C01810=1075.371,111.105,430.185,173.688,24.346,154.284
C01811=1075.364,110.824,430.206,173.687,24.343,154.284
C01812=1075.358,110.542,430.227,173.684,24.341,154.284
C01813=1075.352,110.293,430.246,173.683,24.338,154.283
C01814=1075.347,110.044,430.266,173.681,24.335,154.283
C01815=1075.341,109.795,430.284,173.680,24.333,154.283
C01816=1075.335,109.546,430.303,173.678,24.330,154.283
C01817=1075.329,109.296,430.322,173.676,24.328,154.282
C01818=1075.323,109.047,430.341,173.675,24.325,154.282
C01819=1075.317,108.798,430.360,173.673,24.323,154.282
C01820=1075.312,108.549,430.379,173.671,24.320,154.282
C01821=1075.306,108.300,430.398,173.670,24.318,154.281
C01822=1075.300,108.050,430.417,173.668,24.316,154.281
C01823=1075.294,107.801,430.436,173.666,24.313,154.281
C01824=1075.289,107.552,430.455,173.665,24.311,154.280
C01825=1075.283,107.302,430.473,173.663,24.308,154.280
C01826=1075.277,107.053,430.492,173.661,24.305,154.280
C01827=1075.272,106.804,430.511,173.660,24.303,154.279
C01828=1075.266,106.555,430.530,173.658,24.300,154.279
C01829=1075.260,106.306,430.549,173.656,24.298,154.279
C01830=1075.255,106.056,430.568,173.655,24.295,154.279
C01831=1075.249,105.808,430.587,173.653,24.293,154.278
C01832=1075.243,105.558,430.605,173.651,24.290,154.278
C01833=1075.237,105.309,430.624,173.650,24.287,154.278
C01834=1075.232,105.060,430.643,173.649,24.285,154.277
C01835=1075.226,104.811,430.662,173.646,24.282,154.277
C01836=1075.220,104.561,430.680,173.645,24.280,154.277
C01837=1075.215,104.312,430.699,173.644,24.277,154.277
C01838=1075.209,104.063,430.718,173.642,24.275,154.276
C01839=1075.203,103.814,430.737,173.640,24.272,154.276
C01840=1075.198,103.565,430.756,173.639,24.269,154.276
C01841=1075.192,103.315,430.774,173.637,24.267,154.275
C01842=1075.186,103.066,430.793,173.635,24.264,154.275
C01843=1075.181,102.817,430.812,173.634,24.262,154.275
C01844=1075.175,102.567,430.830,173.632,24.260,154.274
C01845=1075.169,102.318,430.849,173.630,24.256,154.274
C01846=1075.164,102.069,430.868,173.629,24.254,154.274
C01847=1075.158,101.820,430.886,173.627,24.252,154.274
C01848=1075.153,101.571,430.904,173.625,24.249,154.273
C01849=1075.146,101.321,430.923,173.624,24.247,154.273
C01850=1075.141,101.071,430.942,173.623,24.244,154.273
C01851=1075.135,100.823,430.960,173.621,24.241,154.272
C01852=1075.129,100.574,430.979,173.619,24.239,154.272
C01853=1075.123,100.324,430.997,173.618,24.236,154.272
C01854=1075.118,100.075,431.016,173.616,24.234,154.271
C01855=1075.112,99.826,431.035,173.614,24.231,154.271
C01856=1075.106,99.576,431.053,173.613,24.229,154.271
C01857=1075.101,99.327,431.071,173.611,24.227,154.271
C01858=1075.095,99.078,431.089,173.609,24.224,154.270
C01859=1075.089,98.828,431.109,173.608,24.221,154.270
C01860=1075.083,98.580,431.127,173.606,24.219,154.270
C01861=1075.077,98.330,431.145,173.605,24.216,154.269
C01862=1075.072,98.081,431.164,173.603,24.213,154.269
C01863=1075.066,97.832,431.182,173.602,24.211,154.269
C01864=1075.060,97.582,431.201,173.600,24.209,154.269
C01865=1075.054,97.333,431.218,173.598,24.206,154.268
C01866=1075.048,97.084,431.237,173.597,24.203,154.268
C01867=1075.043,96.835,431.255,173.595,24.201,154.268
C01868=1075.037,96.586,431.274,173.593,24.198,154.267
C01869=1075.031,96.336,431.292,173.592,24.196,154.267
C01870=1075.026,96.087,431.311,173.590,24.193,154.267
C01871=1075.019,95.837,431.329,173.589,24.191,154.266
C01872=1075.014,95.589,431.348,173.587,24.188,154.266
C01873=1075.008,95.307,431.368,173.586,24.185,154.266
C01874=1075.001,95.025,431.388,173.583,24.182,154.265
C01875=1074.995,94.744,431.409,173.582,24.180,154.265
C01876=1074.988,94.462,431.430,173.580,24.176,154.265
C01877=1074.983,94.213,431.449,173.579,24.174,154.264
C01878=1074.977,93.963,431.467,173.576,24.171,154.264
C01879=1074.971,93.714,431.484,173.575,24.168,154.264
C01880=1074.965,93.465,431.503,173.574,24.166,154.263
C01881=1074.960,93.216,431.521,173.572,24.164,154.263
C01882=1074.953,92.967,431.540,173.570,24.161,154.263
C01883=1074.949,92.717,431.558,173.569,24.159,154.263
C01884=1074.943,92.468,431.576,173.568,24.156,154.262
C01885=1074.937,92.219,431.594,173.566,24.153,154.262
C01886=1074.931,91.970,431.612,173.564,24.151,154.262
C01887=1074.926,91.720,431.630,173.563,24.148,154.261
C01888=1074.919,91.471,431.649,173.561,24.145,154.261
C01889=1074.914,91.222,431.666,173.559,24.143,154.261
C01890=1074.909,90.972,431.685,173.558,24.140,154.260
C01891=1074.903,90.724,431.703,173.556,24.138,154.260
C01892=1074.897,90.474,431.721,173.555,24.136,154.260
C01893=1074.891,90.225,431.739,173.553,24.132,154.259
C01894=1074.885,89.975,431.757,173.552,24.130,154.259
C01895=1074.879,89.727,431.775,173.550,24.128,154.259
C01896=1074.874,89.477,431.793,173.549,24.125,154.259
C01897=1074.868,89.228,431.811,173.547,24.122,154.258
C01898=1074.862,88.978,431.829,173.545,24.120,154.258
C01899=1074.856,88.729,431.847,173.544,24.117,154.258
C01900=1074.850,88.480,431.865,173.543,24.115,154.257
C01901=1074.844,88.230,431.883,173.541,24.112,154.257
C01902=1074.839,87.981,431.901,173.539,24.110,154.257
C01903=1074.833,87.732,431.919,173.538,24.107,154.257
C01904=1074.827,87.483,431.937,173.537,24.105,154.256
C01905=1074.821,87.234,431.954,173.534,24.102,154.256
C01906=1074.815,86.984,431.972,173.533,24.099,154.256
C01907=1074.810,86.735,431.990,173.532,24.097,154.255
C01908=1074.804,86.485,432.008,173.530,24.095,154.255
C01909=1074.798,86.236,432.027,173.528,24.092,154.255
C01910=1074.792,85.987,432.045,173.527,24.089,154.254
C01911=1074.787,85.738,432.062,173.526,24.087,154.254
C01912=1074.780,85.488,432.080,173.524,24.084,154.254
C01913=1074.775,85.239,432.098,173.522,24.081,154.254
C01914=1074.769,84.989,432.116,173.521,24.079,154.253
C01915=1074.763,84.740,432.133,173.519,24.076,154.253
C01916=1074.758,84.491,432.151,173.518,24.074,154.253
C01917=1074.752,84.241,432.169,173.516,24.071,154.252
C01918=1074.746,83.992,432.186,173.514,24.069,154.252
C01919=1074.740,83.743,432.205,173.513,24.066,154.252
C01920=1074.734,83.494,432.222,173.512,24.063,154.251
C01921=1074.729,83.245,432.240,173.510,24.061,154.251
C01922=1074.723,82.995,432.258,173.508,24.058,154.251
C01923=1074.717,82.746,432.275,173.507,24.056,154.250
C01924=1074.711,82.497,432.293,173.506,24.053,154.250
C01925=1074.705,82.247,432.311,173.504,24.050,154.250
C01926=1074.700,81.998,432.329,173.502,24.048,154.249
C01927=1074.694,81.749,432.346,173.501,24.046,154.249
C01928=1074.688,81.500,432.364,173.500,24.043,154.249
C01929=1074.683,81.251,432.382,173.497,24.040,154.249
C01930=1074.677,81.001,432.400,173.496,24.038,154.248
C01931=1074.671,80.752,432.417,173.495,24.035,154.248
C01932=1074.666,80.503,432.435,173.494,24.032,154.248
C01933=1074.659,80.253,432.453,173.491,24.030,154.247
C01934=1074.654,80.003,432.469,173.490,24.027,154.247
C01935=1074.649,79.754,432.487,173.489,24.024,154.247
C01936=1074.643,79.505,432.505,173.487,24.022,154.246
C01937=1074.636,79.224,432.525,173.485,24.019,154.246
C01938=1074.630,78.942,432.545,173.484,24.016,154.246
C01939=1074.624,78.661,432.565,173.482,24.013,154.245
C01940=1074.617,78.379,432.585,173.481,24.010,154.245
C01941=1074.612,78.129,432.602,173.478,24.007,154.245
C01942=1074.606,77.880,432.620,173.477,24.005,154.244
C01943=1074.600,77.631,432.637,173.476,24.003,154.244
C01944=1074.594,77.382,432.654,173.475,24.000,154.244
C01945=1074.588,77.132,432.672,173.472,23.997,154.243
C01946=1074.582,76.883,432.690,173.471,23.994,154.243
C01947=1074.577,76.634,432.708,173.470,23.992,154.243
C01948=1074.571,76.384,432.725,173.469,23.989,154.242
C01949=1074.564,76.135,432.742,173.467,23.987,154.242
C01950=1074.559,75.886,432.759,173.465,23.984,154.242
C01951=1074.553,75.637,432.777,173.464,23.982,154.242
C01952=1074.547,75.387,432.795,173.462,23.979,154.241
C01953=1074.542,75.137,432.812,173.461,23.976,154.241
C01954=1074.536,74.889,432.829,173.459,23.974,154.241
C01955=1074.530,74.639,432.847,173.457,23.971,154.240
C01956=1074.524,74.390,432.864,173.456,23.969,154.240
C01957=1074.519,74.140,432.881,173.455,23.966,154.240
C01958=1074.512,73.891,432.898,173.454,23.964,154.239
C01959=1074.507,73.642,432.916,173.451,23.961,154.239
C01960=1074.501,73.392,432.933,173.450,23.958,154.239
C01961=1074.496,73.143,432.950,173.449,23.956,154.238
C01962=1074.489,72.894,432.968,173.448,23.953,154.238
C01963=1074.483,72.645,432.985,173.446,23.951,154.238
C01964=1074.478,72.395,433.002,173.444,23.948,154.237
C01965=1074.473,72.146,433.020,173.443,23.945,154.237
C01966=1074.466,71.897,433.037,173.441,23.943,154.237
C01967=1074.461,71.647,433.054,173.440,23.940,154.237
C01968=1074.455,71.398,433.071,173.438,23.937,154.236
C01969=1074.449,71.149,433.088,173.437,23.935,154.236
C01970=1074.443,70.899,433.106,173.435,23.932,154.236
C01971=1074.438,70.650,433.123,173.434,23.930,154.235
C01972=1074.432,70.400,433.140,173.433,23.927,154.235
C01973=1074.426,70.151,433.157,173.431,23.924,154.235
C01974=1074.420,69.902,433.175,173.429,23.922,154.234
C01975=1074.414,69.652,433.191,173.428,23.919,154.234
C01976=1074.408,69.403,433.209,173.427,23.917,154.234
C01977=1074.403,69.154,433.226,173.425,23.914,154.233
C01978=1074.396,68.904,433.243,173.423,23.911,154.233
C01979=1074.391,68.655,433.260,173.422,23.909,154.233
C01980=1074.386,68.405,433.277,173.421,23.906,154.232
C01981=1074.379,68.157,433.294,173.419,23.904,154.232
C01982=1074.374,67.907,433.311,173.418,23.901,154.232
C01983=1074.367,67.658,433.328,173.416,23.898,154.231
C01984=1074.362,67.408,433.345,173.415,23.896,154.231
C01985=1074.356,67.159,433.362,173.413,23.893,154.231
C01986=1074.351,66.910,433.379,173.412,23.891,154.231
C01987=1074.345,66.660,433.397,173.411,23.888,154.230
C01988=1074.339,66.410,433.413,173.408,23.885,154.230
C01989=1074.333,66.161,433.431,173.407,23.883,154.230
C01990=1074.327,65.912,433.447,173.406,23.881,154.229
C01991=1074.322,65.663,433.465,173.405,23.878,154.229
C01992=1074.316,65.414,433.481,173.403,23.875,154.229
C01993=1074.310,65.163,433.498,173.401,23.872,154.228
C01994=1074.304,64.915,433.515,173.400,23.870,154.228
C01995=1074.298,64.665,433.532,173.399,23.867,154.228
C01996=1074.292,64.416,433.549,173.397,23.865,154.227
C01997=1074.287,64.167,433.566,173.396,23.862,154.227
C01998=1074.281,63.918,433.583,173.394,23.860,154.227
C01999=1074.274,63.668,433.599,173.392,23.857,154.226
C02000=1074.269,63.418,433.616,173.391,23.854,154.226
C02001=1074.262,63.137,433.635,173.389,23.852,154.226
C02002=1074.255,62.855,433.654,173.388,23.849,154.226
C02003=1074.248,62.574,433.673,173.386,23.846,154.225
C02004=1074.242,62.293,433.692,173.384,23.843,154.225
C02005=1074.236,62.042,433.709,173.383,23.841,154.225
C02006=1074.230,61.793,433.726,173.382,23.838,154.224
C02007=1074.224,61.544,433.742,173.380,23.835,154.224
C02008=1074.218,61.294,433.759,173.378,23.833,154.224
C02009=1074.212,61.046,433.776,173.377,23.830,154.223
C02010=1074.206,60.796,433.792,173.376,23.828,154.223
C02011=1074.200,60.546,433.809,173.374,23.825,154.223
C02012=1074.194,60.297,433.826,173.373,23.822,154.222
C02013=1074.188,60.048,433.843,173.371,23.820,154.222
C02014=1074.182,59.799,433.859,173.370,23.817,154.222
C02015=1074.177,59.549,433.876,173.368,23.815,154.222
C02016=1074.171,59.300,433.893,173.367,23.812,154.221
C02017=1074.164,59.050,433.909,173.366,23.810,154.221
C02018=1074.159,58.800,433.926,173.364,23.807,154.221
C02019=1074.153,58.551,433.942,173.362,23.804,154.220
C02020=1074.147,58.302,433.959,173.361,23.802,154.220
C02021=1074.141,58.053,433.976,173.360,23.799,154.220
C02022=1074.136,57.803,433.992,173.358,23.797,154.219
C02023=1074.130,57.554,434.009,173.357,23.794,154.219
C02024=1074.124,57.305,434.025,173.355,23.792,154.219
C02025=1074.118,57.055,434.041,173.354,23.789,154.218
C02026=1074.112,56.806,434.059,173.352,23.786,154.218
C02027=1074.106,56.556,434.075,173.351,23.784,154.218
C02028=1074.100,56.307,434.092,173.350,23.781,154.217
C02029=1074.094,56.058,434.108,173.348,23.778,154.217
C02030=1074.089,55.808,434.125,173.346,23.776,154.217
C02031=1074.083,55.559,434.141,173.345,23.773,154.217
C02032=1074.077,55.309,434.157,173.344,23.771,154.216
C02033=1074.070,55.060,434.174,173.342,23.768,154.216
C02034=1074.065,54.811,434.191,173.341,23.766,154.216
C02035=1074.059,54.561,434.207,173.339,23.763,154.215
C02036=1074.053,54.312,434.224,173.338,23.761,154.215
C02037=1074.047,54.063,434.240,173.336,23.758,154.215
C02038=1074.041,53.813,434.256,173.335,23.755,154.214
C02039=1074.036,53.564,434.273,173.334,23.753,154.214
C02040=1074.030,53.314,434.289,173.333,23.750,154.214
C02041=1074.024,53.065,434.305,173.330,23.747,154.213
C02042=1074.018,52.816,434.322,173.329,23.745,154.213
C02043=1074.012,52.566,434.338,173.328,23.742,154.213
C02044=1074.007,52.317,434.355,173.327,23.739,154.212
C02045=1074.001,52.067,434.371,173.325,23.737,154.212
C02046=1073.995,51.818,434.387,173.323,23.734,154.212
C02047=1073.989,51.569,434.404,173.322,23.731,154.211
C02048=1073.983,51.319,434.420,173.321,23.729,154.211
C02049=1073.978,51.070,434.437,173.319,23.727,154.211
C02050=1073.972,50.820,434.453,173.318,23.724,154.210
C02051=1073.966,50.571,434.469,173.317,23.721,154.210
C02052=1073.960,50.322,434.485,173.315,23.718,154.210
C02053=1073.954,50.072,434.502,173.313,23.716,154.210
C02054=1073.949,49.823,434.519,173.312,23.713,154.209
C02055=1073.943,49.573,434.535,173.311,23.711,154.209
C02056=1073.937,49.324,434.551,173.309,23.708,154.209
C02057=1073.931,49.075,434.567,173.308,23.705,154.208
C02058=1073.925,48.825,434.584,173.306,23.703,154.208
C02059=1073.919,48.576,434.600,173.305,23.700,154.208
C02060=1073.914,48.327,434.616,173.304,23.697,154.207
C02061=1073.909,48.078,434.633,173.302,23.695,154.207
C02062=1073.903,47.828,434.648,173.301,23.693,154.207
C02063=1073.897,47.578,434.664,173.300,23.690,154.206
C02064=1073.891,47.329,434.681,173.298,23.687,154.206
C02065=1073.885,47.047,434.699,173.296,23.684,154.206
C02066=1073.878,46.766,434.717,173.295,23.681,154.205
C02067=1073.871,46.483,434.736,173.293,23.678,154.205
C02068=1073.865,46.202,434.754,173.292,23.675,154.205
C02069=1073.859,45.952,434.770,173.291,23.673,154.204
C02070=1073.854,45.703,434.787,173.288,23.669,154.204
C02071=1073.848,45.454,434.803,173.287,23.667,154.204
C02072=1073.843,45.204,434.818,173.286,23.664,154.203
C02073=1073.837,44.955,434.835,173.285,23.662,154.203
C02074=1073.831,44.705,434.851,173.283,23.659,154.203
C02075=1073.825,44.456,434.867,173.282,23.656,154.202
C02076=1073.819,44.206,434.883,173.280,23.654,154.202
C02077=1073.813,43.957,434.899,173.279,23.651,154.202
C02078=1073.808,43.708,434.915,173.278,23.648,154.201
C02079=1073.802,43.459,434.931,173.276,23.646,154.201
C02080=1073.796,43.209,434.947,173.275,23.644,154.201
C02081=1073.790,42.959,434.963,173.274,23.641,154.200
C02082=1073.785,42.710,434.979,173.272,23.638,154.200
C02083=1073.779,42.461,434.995,173.270,23.635,154.200
C02084=1073.773,42.211,435.011,173.269,23.633,154.199
C02085=1073.767,41.961,435.027,173.268,23.631,154.199
C02086=1073.761,41.712,435.043,173.266,23.628,154.199
C02087=1073.756,41.463,435.059,173.265,23.625,154.198
C02088=1073.750,41.213,435.075,173.264,23.623,154.198
C02089=1073.743,40.964,435.090,173.262,23.620,154.198
C02090=1073.738,40.714,435.106,173.260,23.617,154.198
C02091=1073.732,40.465,435.122,173.259,23.615,154.197
C02092=1073.726,40.216,435.139,173.258,23.612,154.197
C02093=1073.721,39.966,435.154,173.257,23.609,154.197
C02094=1073.715,39.717,435.170,173.255,23.607,154.196
C02095=1073.709,39.467,435.186,173.254,23.605,154.196
C02096=1073.703,39.218,435.202,173.252,23.601,154.196
C02097=1073.697,38.968,435.218,173.251,23.599,154.195
C02098=1073.691,38.719,435.233,173.249,23.596,154.195
C02099=1073.686,38.470,435.249,173.248,23.594,154.195
C02100=1073.680,38.220,435.264,173.247,23.591,154.194
C02101=1073.674,37.971,435.281,173.246,23.589,154.194
C02102=1073.668,37.721,435.297,173.244,23.586,154.194
C02103=1073.662,37.471,435.312,173.242,23.584,154.194
C02104=1073.656,37.222,435.328,173.241,23.581,154.193
C02105=1073.651,36.973,435.343,173.240,23.578,154.193
C02106=1073.645,36.724,435.360,173.238,23.576,154.193
C02107=1073.638,36.474,435.375,173.237,23.573,154.192
C02108=1073.632,36.225,435.391,173.236,23.570,154.192
C02109=1073.627,35.975,435.406,173.234,23.568,154.192
C02110=1073.621,35.726,435.422,173.232,23.565,154.191
C02111=1073.615,35.476,435.437,173.231,23.563,154.191
C02112=1073.609,35.227,435.453,173.230,23.560,154.191
C02113=1073.603,34.977,435.469,173.229,23.558,154.190
C02114=1073.597,34.728,435.485,173.227,23.555,154.190
C02115=1073.592,34.479,435.500,173.226,23.553,154.190
C02116=1073.586,34.229,435.516,173.224,23.550,154.189
C02117=1073.579,33.980,435.531,173.222,23.548,154.189
C02118=1073.574,33.730,435.547,173.221,23.545,154.189
C02119=1073.568,33.480,435.563,173.220,23.542,154.189
C02120=1073.562,33.232,435.577,173.219,23.540,154.188
C02121=1073.556,32.982,435.594,173.217,23.537,154.188
C02122=1073.550,32.732,435.609,173.216,23.534,154.188
C02123=1073.544,32.483,435.624,173.214,23.532,154.187
C02124=1073.539,32.234,435.640,173.213,23.529,154.187
C02125=1073.533,31.984,435.656,173.211,23.527,154.187
C02126=1073.526,31.735,435.671,173.210,23.524,154.186
C02127=1073.521,31.485,435.687,173.209,23.521,154.186
C02128=1073.516,31.236,435.702,173.208,23.519,154.186
C02129=1073.508,30.954,435.719,173.206,23.516,154.185
C02130=1073.502,30.672,435.737,173.204,23.513,154.185
C02131=1073.495,30.390,435.754,173.203,23.510,154.185
C02132=1073.489,30.108,435.772,173.201,23.507,154.184
C02133=1073.483,29.859,435.787,173.200,23.505,154.184
C02134=1073.477,29.609,435.803,173.199,23.502,154.184
C02135=1073.471,29.360,435.818,173.197,23.499,154.183
C02136=1073.465,29.110,435.833,173.196,23.497,154.183
C02137=1073.459,28.861,435.850,173.194,23.494,154.183
C02138=1073.453,28.612,435.864,173.193,23.492,154.182
C02139=1073.448,28.362,435.880,173.191,23.489,154.182
C02140=1073.441,28.112,435.895,173.190,23.486,154.182
C02141=1073.436,27.864,435.911,173.189,23.484,154.182
C02142=1073.430,27.614,435.926,173.188,23.482,154.181
C02143=1073.424,27.364,435.941,173.186,23.479,154.181
C02144=1073.418,27.115,435.956,173.185,23.477,154.181
C02145=1073.413,26.865,435.971,173.183,23.473,154.180
C02146=1073.406,26.616,435.987,173.182,23.471,154.180
C02147=1073.400,26.366,436.002,173.180,23.469,154.180
C02148=1073.394,26.117,436.017,173.179,23.466,154.179
C02149=1073.389,25.867,436.033,173.178,23.464,154.179
C02150=1073.382,25.618,436.047,173.176,23.461,154.179
C02151=1073.376,25.369,436.063,173.175,23.458,154.178
C02152=1073.371,25.119,436.078,173.173,23.456,154.178
C02153=1073.364,24.870,436.093,173.172,23.453,154.178
C02154=1073.359,24.620,436.108,173.170,23.451,154.178
C02155=1073.353,24.371,436.123,173.169,23.448,154.177
C02156=1073.347,24.121,436.139,173.168,23.445,154.177
C02157=1073.342,23.872,436.153,173.167,23.443,154.177
C02158=1073.335,23.623,436.169,173.165,23.441,154.176
C02159=1073.329,23.373,436.185,173.164,23.438,154.176
C02160=1073.323,23.124,436.199,173.162,23.435,154.176
C02161=1073.318,22.874,436.215,173.161,23.433,154.176
C02162=1073.311,22.624,436.230,173.159,23.430,154.175
C02163=1073.306,22.375,436.245,173.158,23.428,154.175
C02164=1073.300,22.125,436.260,173.157,23.425,154.175
C02165=1073.294,21.876,436.274,173.156,23.423,154.174
C02166=1073.289,21.626,436.290,173.154,23.420,154.174
C02167=1073.282,21.377,436.305,173.153,23.417,154.174
C02168=1073.277,21.128,436.320,173.151,23.415,154.173
C02169=1073.271,20.878,436.335,173.150,23.412,154.173
C02170=1073.264,20.628,436.350,173.148,23.410,154.173
C02171=1073.259,20.379,436.365,173.147,23.407,154.172
C02172=1073.253,20.129,436.380,173.146,23.404,154.172
C02173=1073.247,19.880,436.395,173.145,23.402,154.172
C02174=1073.241,19.630,436.410,173.143,23.400,154.172
C02175=1073.235,19.381,436.425,173.142,23.397,154.171
C02176=1073.229,19.132,436.440,173.140,23.394,154.171
C02177=1073.223,18.882,436.455,173.138,23.392,154.171
C02178=1073.218,18.633,436.470,173.137,23.390,154.170
C02179=1073.211,18.383,436.485,173.136,23.387,154.170
C02180=1073.205,18.134,436.500,173.135,23.384,154.170
C02181=1073.200,17.884,436.515,173.133,23.382,154.169
C02182=1073.194,17.635,436.530,173.132,23.379,154.169
C02183=1073.188,17.386,436.544,173.131,23.377,154.169
C02184=1073.182,17.136,436.559,173.129,23.374,154.169
C02185=1073.176,16.887,436.575,173.127,23.372,154.168
C02186=1073.170,16.637,436.590,173.126,23.369,154.168
C02187=1073.165,16.387,436.603,173.125,23.366,154.168
C02188=1073.158,16.138,436.618,173.124,23.364,154.167
C02189=1073.153,15.888,436.634,173.122,23.362,154.167
C02190=1073.147,15.639,436.648,173.121,23.359,154.167
C02191=1073.140,15.389,436.663,173.120,23.357,154.167
C02192=1073.135,15.140,436.678,173.118,23.353,154.166
C02193=1073.128,14.860,436.695,173.116,23.351,154.166
C02194=1073.121,14.580,436.711,173.115,23.348,154.165
C02195=1073.115,14.299,436.728,173.113,23.345,154.165
C02196=1073.108,14.018,436.745,173.112,23.342,154.165
C02197=1073.102,13.769,436.759,173.111,23.340,154.165
C02198=1073.096,13.519,436.773,173.109,23.337,154.164
C02199=1073.090,13.270,436.788,173.108,23.335,154.164
C02200=1073.084,13.021,436.803,173.106,23.332,154.164
C02201=1073.078,12.770,436.818,173.105,23.330,154.163
C02202=1073.073,12.521,436.832,173.103,23.327,154.163
C02203=1073.066,12.271,436.847,173.102,23.325,154.163
C02204=1073.060,12.022,436.862,173.101,23.323,154.163
C02205=1073.054,11.772,436.876,173.099,23.320,154.162
C02206=1073.049,11.523,436.891,173.098,23.318,154.162
C02207=1073.042,11.274,436.906,173.097,23.315,154.162
C02208=1073.036,11.025,436.920,173.096,23.313,154.161
C02209=1073.030,10.774,436.934,173.093,23.310,154.161
C02210=1073.025,10.525,436.949,173.092,23.308,154.161
C02211=1073.018,10.276,436.964,173.091,23.305,154.161
C02212=1073.013,10.026,436.978,173.090,23.303,154.160
C02213=1073.006,9.776,436.993,173.088,23.300,154.160
C02214=1073.001,9.528,437.007,173.087,23.298,154.160
C02215=1072.994,9.277,437.022,173.086,23.296,154.159
C02216=1072.989,9.028,437.036,173.084,23.293,154.159
C02217=1072.982,8.779,437.051,173.082,23.290,154.159
C02218=1072.977,8.529,437.065,173.081,23.287,154.159
C02219=1072.970,8.279,437.080,173.080,23.285,154.158
C02220=1072.965,8.030,437.095,173.078,23.283,154.158
C02221=1072.959,7.780,437.109,173.077,23.280,154.158
C02222=1072.953,7.531,437.123,173.076,23.278,154.157
C02223=1072.946,7.282,437.138,173.075,23.275,154.157
C02224=1072.941,7.032,437.152,173.073,23.273,154.157
C02225=1072.935,6.782,437.167,173.072,23.270,154.157
C02226=1072.929,6.533,437.181,173.070,23.268,154.156
C02227=1072.923,6.283,437.196,173.069,23.265,154.156
C02228=1072.917,6.034,437.210,173.067,23.263,154.156
C02229=1072.911,5.785,437.224,173.066,23.260,154.155
C02230=1072.905,5.535,437.239,173.065,23.258,154.155
C02231=1072.900,5.285,437.253,173.063,23.255,154.155
C02232=1072.893,5.036,437.268,173.062,23.253,154.155
C02233=1072.888,4.786,437.282,173.061,23.251,154.154
C02234=1072.881,4.537,437.296,173.059,23.248,154.154
C02235=1072.875,4.287,437.310,173.057,23.245,154.154
C02236=1072.869,4.038,437.325,173.056,23.242,154.153
C02237=1072.863,3.788,437.339,173.055,23.240,154.153
C02238=1072.857,3.539,437.354,173.054,23.238,154.153
C02239=1072.852,3.289,437.367,173.052,23.235,154.153
C02240=1072.846,3.040,437.382,173.051,23.233,154.152
C02241=1072.840,2.790,437.396,173.050,23.230,154.152
C02242=1072.834,2.541,437.411,173.049,23.228,154.152
C02243=1072.828,2.291,437.425,173.046,23.225,154.151
C02244=1072.823,2.041,437.439,173.045,23.223,154.151
C02245=1072.816,1.792,437.454,173.044,23.220,154.151
C02246=1072.811,1.542,437.468,173.042,23.218,154.151
C02247=1072.805,1.293,437.482,173.041,23.215,154.150
C02248=1072.798,1.043,437.496,173.040,23.213,154.150
C02249=1072.793,0.794,437.511,173.039,23.211,154.150
C02250=1072.787,0.545,437.524,173.037,23.208,154.149
C02251=1072.781,0.294,437.539,173.036,23.206,154.149
C02252=1072.775,0.045,437.553,173.034,23.203,154.149
C02253=1072.770,-0.204,437.567,173.033,23.200,154.149
C02254=1072.764,-0.454,437.581,173.031,23.198,154.148
C02255=1072.758,-0.703,437.596,173.030,23.196,154.148
C02256=1072.752,-0.953,437.610,173.029,23.193,154.148
C02257=1072.745,-1.231,437.626,173.028,23.190,154.147
C02258=1072.739,-1.510,437.641,173.025,23.187,154.147
C02259=1072.732,-1.788,437.657,173.024,23.184,154.147
C02260=1072.726,-2.067,437.673,173.023,23.182,154.146
C02261=1072.720,-2.316,437.687,173.021,23.179,154.146
C02262=1072.714,-2.565,437.701,173.020,23.177,154.146
C02263=1072.709,-2.815,437.715,173.018,23.174,154.146
C02264=1072.702,-3.065,437.730,173.017,23.172,154.145
C02265=1072.697,-3.314,437.743,173.016,23.170,154.145
C02266=1072.691,-3.564,437.757,173.014,23.167,154.145
C02267=1072.685,-3.814,437.771,173.013,23.165,154.145
C02268=1072.679,-4.063,437.785,173.012,23.162,154.144
C02269=1072.673,-4.312,437.799,173.011,23.160,154.144
C02270=1072.667,-4.562,437.813,173.009,23.157,154.144
C02271=1072.661,-4.812,437.827,173.007,23.155,154.143
C02272=1072.655,-5.061,437.841,173.006,23.152,154.143
C02273=1072.648,-5.311,437.855,173.004,23.150,154.143
C02274=1072.643,-5.560,437.869,173.003,23.148,154.143
C02275=1072.637,-5.810,437.882,173.002,23.145,154.142
C02276=1072.631,-6.060,437.896,173.001,23.143,154.142
C02277=1072.625,-6.309,437.911,172.999,23.141,154.142
C02278=1072.619,-6.558,437.924,172.998,23.138,154.142
C02279=1072.613,-6.808,437.938,172.997,23.136,154.141
C02280=1072.606,-7.058,437.952,172.995,23.133,154.141
C02281=1072.601,-7.307,437.966,172.993,23.130,154.141
C02282=1072.595,-7.557,437.980,172.992,23.129,154.141
C02283=1072.588,-7.806,437.994,172.991,23.126,154.140
C02284=1072.583,-8.056,438.008,172.989,23.124,154.140
C02285=1072.577,-8.305,438.021,172.988,23.121,154.140
C02286=1072.571,-8.555,438.035,172.987,23.119,154.140
C02287=1072.565,-8.805,438.049,172.985,23.116,154.139
C02288=1072.559,-9.054,438.062,172.984,23.114,154.139
C02289=1072.553,-9.304,438.076,172.982,23.111,154.139
C02290=1072.547,-9.553,438.089,172.981,23.109,154.138
C02291=1072.541,-9.803,438.104,172.979,23.107,154.138
C02292=1072.535,-10.053,438.117,172.978,23.104,154.138
C02293=1072.529,-10.302,438.131,172.977,23.102,154.138
C02294=1072.524,-10.551,438.145,172.975,23.100,154.137
C02295=1072.517,-10.800,438.159,172.974,23.097,154.137
C02296=1072.511,-11.051,438.173,172.973,23.095,154.137
C02297=1072.505,-11.300,438.186,172.972,23.092,154.137
C02298=1072.500,-11.549,438.200,172.969,23.089,154.136
C02299=1072.493,-11.799,438.213,172.968,23.088,154.136
C02300=1072.488,-12.048,438.227,172.967,23.085,154.136
C02301=1072.481,-12.298,438.241,172.965,23.083,154.136
C02302=1072.476,-12.548,438.255,172.964,23.080,154.135
C02303=1072.470,-12.797,438.269,172.963,23.078,154.135
C02304=1072.464,-13.047,438.282,172.962,23.075,154.135
C02305=1072.458,-13.296,438.296,172.960,23.073,154.135
C02306=1072.452,-13.545,438.309,172.959,23.071,154.134
C02307=1072.446,-13.796,438.323,172.958,23.069,154.134
C02308=1072.440,-14.045,438.336,172.955,23.066,154.134
C02309=1072.435,-14.295,438.350,172.954,23.063,154.134
C02310=1072.429,-14.544,438.363,172.953,23.061,154.133
C02311=1072.423,-14.794,438.377,172.952,23.059,154.133
C02312=1072.417,-15.043,438.390,172.950,23.056,154.133
C02313=1072.411,-15.293,438.404,172.949,23.054,154.133
C02314=1072.405,-15.543,438.418,172.948,23.052,154.132
C02315=1072.398,-15.792,438.431,172.946,23.049,154.132
C02316=1072.393,-16.042,438.445,172.945,23.047,154.132
C02317=1072.387,-16.291,438.458,172.944,23.045,154.132
C02318=1072.380,-16.540,438.471,172.941,23.042,154.131
C02319=1072.374,-16.791,438.485,172.940,23.040,154.131
C02320=1072.369,-17.040,438.498,172.939,23.037,154.131
C02321=1072.362,-17.317,438.512,172.938,23.035,154.130
C02322=1072.355,-17.594,438.528,172.936,23.032,154.130
C02323=1072.349,-17.871,438.542,172.934,23.030,154.130
C02324=1072.342,-18.148,438.557,172.933,23.027,154.130
C02325=1072.336,-18.397,438.571,172.932,23.025,154.130
C02326=1072.330,-18.646,438.584,172.930,23.023,154.129
C02327=1072.324,-18.896,438.598,172.929,23.020,154.129
C02328=1072.318,-19.145,438.612,172.927,23.018,154.129
C02329=1072.312,-19.395,438.624,172.925,23.016,154.129
C02330=1072.306,-19.644,438.637,172.924,23.013,154.128
C02331=1072.301,-19.894,438.651,172.923,23.011,154.128
C02332=1072.294,-20.144,438.665,172.922,23.008,154.128
C02333=1072.288,-20.394,438.678,172.920,23.007,154.128
C02334=1072.282,-20.643,438.691,172.919,23.004,154.127
C02335=1072.276,-20.893,438.705,172.918,23.002,154.127
C02336=1072.270,-21.142,438.718,172.916,23.000,154.127
C02337=1072.264,-21.392,438.730,172.915,22.997,154.127
C02338=1072.259,-21.641,438.744,172.913,22.995,154.126
C02339=1072.252,-21.891,438.758,172.911,22.992,154.126
C02340=1072.246,-22.141,438.770,172.910,22.990,154.126
C02341=1072.240,-22.390,438.783,172.909,22.988,154.126
C02342=1072.235,-22.639,438.797,172.907,22.985,154.125
C02343=1072.229,-22.889,438.811,172.906,22.983,154.125
C02344=1072.222,-23.139,438.823,172.905,22.981,154.125
C02345=1072.216,-23.389,438.837,172.903,22.979,154.125
C02346=1072.210,-23.638,438.851,172.902,22.976,154.124
C02347=1072.204,-23.888,438.863,172.901,22.974,154.124
C02348=1072.198,-24.137,438.876,172.899,22.971,154.124
C02349=1072.192,-24.387,438.889,172.897,22.969,154.124
C02350=1072.187,-24.637,438.903,172.896,22.967,154.124
C02351=1072.181,-24.886,438.916,172.895,22.965,154.123
C02352=1072.175,-25.136,438.929,172.893,22.962,154.123
C02353=1072.168,-25.385,438.942,172.892,22.960,154.123
C02354=1072.163,-25.635,438.956,172.891,22.958,154.123
C02355=1072.157,-25.885,438.968,172.889,22.955,154.122
C02356=1072.151,-26.134,438.982,172.888,22.954,154.122
C02357=1072.145,-26.384,438.994,172.887,22.951,154.122
C02358=1072.140,-26.633,439.008,172.884,22.948,154.122
C02359=1072.134,-26.883,439.021,172.883,22.946,154.121
C02360=1072.127,-27.132,439.034,172.882,22.944,154.121
C02361=1072.121,-27.382,439.047,172.881,22.942,154.121
C02362=1072.115,-27.632,439.060,172.879,22.940,154.121
C02363=1072.109,-27.881,439.073,172.878,22.937,154.120
C02364=1072.103,-28.131,439.086,172.876,22.935,154.120
C02365=1072.097,-28.380,439.099,172.875,22.933,154.120
C02366=1072.091,-28.630,439.111,172.874,22.931,154.120
C02367=1072.085,-28.879,439.125,172.872,22.929,154.120
C02368=1072.079,-29.129,439.137,172.870,22.926,154.119
C02369=1072.073,-29.378,439.150,172.869,22.924,154.119
C02370=1072.067,-29.628,439.163,172.868,22.921,154.119
C02371=1072.061,-29.877,439.176,172.866,22.920,154.119
C02372=1072.055,-30.127,439.189,172.865,22.917,154.118
C02373=1072.048,-30.377,439.202,172.863,22.915,154.118
C02374=1072.043,-30.626,439.215,172.862,22.913,154.118
C02375=1072.037,-30.876,439.227,172.861,22.911,154.118
C02376=1072.030,-31.126,439.240,172.859,22.908,154.118
C02377=1072.024,-31.376,439.253,172.858,22.907,154.117
C02378=1072.018,-31.625,439.266,172.857,22.904,154.117
C02379=1072.012,-31.875,439.279,172.854,22.902,154.117
C02380=1072.006,-32.124,439.292,172.853,22.899,154.117
C02381=1072.000,-32.374,439.305,172.852,22.897,154.117
C02382=1071.994,-32.624,439.317,172.850,22.895,154.116
C02383=1071.988,-32.873,439.330,172.849,22.893,154.116
C02384=1071.982,-33.123,439.343,172.848,22.891,154.116
C02385=1071.976,-33.399,439.357,172.846,22.888,154.116
C02386=1071.970,-33.675,439.372,172.844,22.885,154.115
C02387=1071.963,-33.950,439.385,172.843,22.884,154.115
C02388=1071.956,-34.227,439.400,172.842,22.881,154.115
C02389=1071.950,-34.476,439.412,172.840,22.879,154.115
C02390=1071.944,-34.726,439.425,172.839,22.877,154.115
C02391=1071.938,-34.976,439.438,172.837,22.874,154.114
C02392=1071.932,-35.226,439.451,172.835,22.872,154.114
C02393=1071.926,-35.475,439.463,172.834,22.870,154.114
C02394=1071.921,-35.724,439.476,172.833,22.868,154.114
C02395=1071.915,-35.974,439.489,172.831,22.865,154.113
C02396=1071.909,-36.224,439.501,172.830,22.863,154.113
C02397=1071.903,-36.473,439.515,172.829,22.861,154.113
C02398=1071.897,-36.723,439.527,172.827,22.859,154.113
C02399=1071.890,-36.972,439.539,172.826,22.857,154.113
C02400=1071.884,-37.222,439.552,172.824,22.855,154.112
C02401=1071.879,-37.471,439.564,172.823,22.852,154.112
C02402=1071.873,-37.721,439.577,172.821,22.850,154.112
C02403=1071.867,-37.971,439.590,172.819,22.848,154.112
C02404=1071.861,-38.221,439.602,172.818,22.846,154.112
C02405=1071.855,-38.470,439.615,172.817,22.844,154.111
C02406=1071.849,-38.720,439.628,172.816,22.841,154.111
C02407=1071.843,-38.970,439.641,172.814,22.839,154.111
C02408=1071.836,-39.219,439.652,172.813,22.837,154.111
C02409=1071.831,-39.468,439.665,172.811,22.835,154.111
C02410=1071.825,-39.718,439.677,172.810,22.833,154.110
C02411=1071.819,-39.967,439.691,172.809,22.831,154.110
C02412=1071.812,-40.217,439.702,172.807,22.829,154.110
C02413=1071.806,-40.467,439.715,172.805,22.826,154.110
C02414=1071.800,-40.717,439.728,172.804,22.824,154.110
C02415=1071.794,-40.967,439.740,172.802,22.822,154.109
C02416=1071.788,-41.216,439.752,172.801,22.820,154.109
C02417=1071.782,-41.465,439.764,172.800,22.818,154.109
C02418=1071.776,-41.715,439.778,172.798,22.816,154.109
C02419=1071.770,-41.965,439.790,172.797,22.814,154.109
C02420=1071.764,-42.214,439.802,172.795,22.812,154.108
C02421=1071.758,-42.464,439.815,172.794,22.810,154.108
C02422=1071.752,-42.714,439.827,172.793,22.808,154.108
C02423=1071.747,-42.963,439.839,172.791,22.805,154.108
C02424=1071.740,-43.213,439.851,172.789,22.803,154.108
C02425=1071.734,-43.463,439.864,172.788,22.801,154.108
C02426=1071.728,-43.712,439.876,172.786,22.799,154.107
C02427=1071.721,-43.962,439.888,172.785,22.797,154.107
C02428=1071.716,-44.211,439.901,172.783,22.795,154.107
C02429=1071.710,-44.461,439.913,172.782,22.793,154.107
C02430=1071.704,-44.711,439.925,172.781,22.791,154.107
C02431=1071.698,-44.961,439.938,172.779,22.789,154.106
C02432=1071.692,-45.210,439.950,172.778,22.787,154.106
C02433=1071.686,-45.460,439.962,172.776,22.785,154.106
C02434=1071.680,-45.709,439.974,172.775,22.782,154.106
C02435=1071.674,-45.959,439.987,172.774,22.781,154.106
C02436=1071.668,-46.209,439.999,172.771,22.778,154.106
C02437=1071.662,-46.458,440.011,172.770,22.776,154.105
C02438=1071.656,-46.708,440.024,172.769,22.774,154.105
C02439=1071.650,-46.958,440.036,172.767,22.772,154.105
C02440=1071.644,-47.207,440.048,172.766,22.770,154.105
C02441=1071.638,-47.456,440.060,172.765,22.768,154.105
C02442=1071.632,-47.706,440.073,172.763,22.766,154.104
C02443=1071.626,-47.956,440.085,172.762,22.764,154.104
C02444=1071.620,-48.206,440.097,172.760,22.762,154.104
C02445=1071.614,-48.455,440.110,172.759,22.759,154.104
C02446=1071.608,-48.704,440.121,172.758,22.758,154.104
C02447=1071.602,-48.954,440.134,172.756,22.756,154.104
C02448=1071.597,-49.203,440.146,172.755,22.754,154.103
C02449=1071.590,-49.480,440.159,172.753,22.751,154.103
C02450=1071.582,-49.757,440.173,172.751,22.749,154.103
C02451=1071.577,-50.033,440.186,172.750,22.747,154.103
C02452=1071.570,-50.310,440.199,172.748,22.744,154.103
C02453=1071.564,-50.560,440.212,172.746,22.742,154.103
C02454=1071.558,-50.809,440.223,172.745,22.741,154.102
C02455=1071.551,-51.058,440.235,172.743,22.739,154.102
C02456=1071.545,-51.308,440.248,172.742,22.736,154.102
C02457=1071.539,-51.558,440.260,172.741,22.734,154.102
C02458=1071.533,-51.808,440.272,172.739,22.732,154.102
C02459=1071.527,-52.057,440.283,172.738,22.730,154.102
C02460=1071.520,-52.307,440.295,172.736,22.729,154.101
C02461=1071.514,-52.556,440.308,172.735,22.727,154.101
C02462=1071.508,-52.806,440.320,172.733,22.725,154.101
C02463=1071.502,-53.056,440.331,172.731,22.722,154.101
C02464=1071.496,-53.305,440.343,172.730,22.721,154.101
C02465=1071.489,-53.555,440.355,172.728,22.719,154.101
C02466=1071.483,-53.804,440.367,172.727,22.717,154.101
C02467=1071.478,-54.054,440.379,172.725,22.715,154.100
C02468=1071.471,-54.304,440.391,172.724,22.713,154.100
C02469=1071.464,-54.553,440.403,172.723,22.711,154.100
C02470=1071.459,-54.803,440.415,172.721,22.709,154.100
C02471=1071.453,-55.053,440.426,172.720,22.707,154.100
C02472=1071.446,-55.302,440.438,172.718,22.705,154.100
C02473=1071.441,-55.552,440.450,172.717,22.703,154.099
C02474=1071.434,-55.801,440.462,172.715,22.702,154.099
C02475=1071.428,-56.051,440.473,172.714,22.700,154.099
C02476=1071.422,-56.301,440.486,172.713,22.698,154.099
C02477=1071.416,-56.550,440.497,172.710,22.695,154.099
C02478=1071.410,-56.800,440.509,172.709,22.694,154.099
C02479=1071.404,-57.050,440.521,172.707,22.692,154.099
C02480=1071.398,-57.299,440.533,172.706,22.690,154.098
C02481=1071.391,-57.549,440.544,172.704,22.688,154.098
C02482=1071.385,-57.799,440.557,172.703,22.686,154.098
C02483=1071.379,-58.048,440.568,172.702,22.684,154.098
C02484=1071.373,-58.298,440.579,172.700,22.682,154.098
C02485=1071.368,-58.547,440.592,172.699,22.680,154.098
C02486=1071.361,-58.798,440.603,172.697,22.678,154.098
C02487=1071.355,-59.047,440.615,172.696,22.676,154.097
C02488=1071.349,-59.296,440.626,172.694,22.675,154.097
C02489=1071.343,-59.547,440.638,172.693,22.673,154.097
C02490=1071.336,-59.796,440.650,172.691,22.671,154.097
C02491=1071.331,-60.046,440.661,172.690,22.669,154.097
C02492=1071.325,-60.295,440.674,172.688,22.667,154.097
C02493=1071.319,-60.544,440.685,172.686,22.665,154.097
C02494=1071.312,-60.795,440.697,172.685,22.663,154.097
C02495=1071.306,-61.044,440.709,172.683,22.661,154.096
C02496=1071.301,-61.294,440.720,172.682,22.660,154.096
C02497=1071.294,-61.543,440.732,172.681,22.658,154.096
C02498=1071.288,-61.793,440.743,172.679,22.656,154.096
C02499=1071.282,-62.043,440.755,172.678,22.654,154.096
C02500=1071.277,-62.292,440.766,172.676,22.652,154.096
C02501=1071.270,-62.542,440.778,172.675,22.651,154.096
C02502=1071.264,-62.792,440.789,172.673,22.649,154.095
C02503=1071.258,-63.041,440.802,172.672,22.647,154.095
C02504=1071.252,-63.291,440.813,172.670,22.645,154.095
C02505=1071.246,-63.540,440.824,172.669,22.643,154.095
C02506=1071.240,-63.791,440.836,172.668,22.641,154.095
C02507=1071.234,-64.040,440.848,172.666,22.639,154.095
C02508=1071.228,-64.290,440.859,172.664,22.637,154.095
C02509=1071.222,-64.539,440.871,172.662,22.635,154.095
C02510=1071.216,-64.789,440.882,172.661,22.634,154.094
C02511=1071.210,-65.038,440.893,172.659,22.632,154.094
C02512=1071.204,-65.288,440.905,172.658,22.630,154.094
C02513=1071.197,-65.566,440.918,172.656,22.628,154.094
C02514=1071.190,-65.844,440.931,172.655,22.626,154.094
C02515=1071.184,-66.121,440.944,172.653,22.624,154.094
C02516=1071.177,-66.399,440.956,172.651,22.622,154.094
C02517=1071.171,-66.649,440.968,172.650,22.620,154.093
C02518=1071.165,-66.898,440.978,172.648,22.618,154.093
C02519=1071.159,-67.148,440.991,172.647,22.616,154.093
C02520=1071.153,-67.398,441.002,172.646,22.614,154.093
C02521=1071.147,-67.648,441.013,172.644,22.613,154.093
C02522=1071.141,-67.897,441.025,172.643,22.611,154.093
C02523=1071.135,-68.147,441.036,172.641,22.609,154.093
C02524=1071.130,-68.397,441.047,172.640,22.607,154.093
C02525=1071.123,-68.646,441.059,172.638,22.605,154.092
C02526=1071.117,-68.896,441.070,172.637,22.604,154.092
C02527=1071.111,-69.146,441.082,172.634,22.602,154.092
C02528=1071.105,-69.395,441.093,172.633,22.600,154.092
C02529=1071.100,-69.645,441.105,172.631,22.598,154.092
C02530=1071.094,-69.895,441.116,172.630,22.596,154.092
C02531=1071.088,-70.144,441.127,172.628,22.594,154.092
C02532=1071.081,-70.394,441.139,172.627,22.593,154.092
C02533=1071.075,-70.643,441.150,172.626,22.591,154.092
C02534=1071.069,-70.894,441.161,172.624,22.589,154.091
C02535=1071.064,-71.143,441.173,172.623,22.587,154.091
C02536=1071.058,-71.392,441.184,172.621,22.585,154.091
C02537=1071.052,-71.642,441.195,172.620,22.584,154.091
C02538=1071.046,-71.892,441.206,172.618,22.582,154.091
C02539=1071.039,-72.142,441.218,172.617,22.580,154.091
C02540=1071.034,-72.391,441.229,172.615,22.578,154.091
C02541=1071.028,-72.641,441.240,172.614,22.576,154.091
C02542=1071.022,-72.891,441.252,172.612,22.575,154.091
C02543=1071.017,-73.141,441.262,172.611,22.573,154.090
C02544=1071.010,-73.390,441.274,172.609,22.571,154.090
C02545=1071.004,-73.640,441.285,172.608,22.569,154.090
C02546=1070.998,-73.889,441.296,172.606,22.568,154.090
C02547=1070.992,-74.139,441.307,172.605,22.566,154.090
C02548=1070.986,-74.389,441.318,172.603,22.564,154.090
C02549=1070.980,-74.639,441.329,172.601,22.563,154.090
C02550=1070.974,-74.888,441.340,172.600,22.561,154.090
C02551=1070.968,-75.137,441.352,172.598,22.559,154.090
C02552=1070.962,-75.387,441.363,172.597,22.557,154.090
C02553=1070.956,-75.637,441.374,172.595,22.556,154.090
C02554=1070.950,-75.887,441.385,172.594,22.554,154.089
C02555=1070.944,-76.137,441.396,172.592,22.552,154.089
C02556=1070.938,-76.386,441.407,172.591,22.551,154.089
C02557=1070.931,-76.636,441.418,172.589,22.549,154.089
C02558=1070.925,-76.886,441.429,172.587,22.548,154.089
C02559=1070.919,-77.136,441.440,172.586,22.546,154.089
C02560=1070.913,-77.385,441.451,172.584,22.544,154.089
C02561=1070.907,-77.634,441.462,172.583,22.542,154.089
C02562=1070.901,-77.884,441.474,172.581,22.541,154.089
C02563=1070.895,-78.134,441.484,172.580,22.539,154.089
C02564=1070.890,-78.383,441.495,172.578,22.538,154.089
C02565=1070.883,-78.633,441.507,172.577,22.536,154.088
C02566=1070.877,-78.883,441.517,172.575,22.535,154.088
C02567=1070.872,-79.132,441.528,172.574,22.533,154.088
C02568=1070.865,-79.382,441.539,172.572,22.531,154.088
C02569=1070.859,-79.632,441.550,172.571,22.529,154.088
C02570=1070.853,-79.881,441.561,172.569,22.528,154.088
C02571=1070.847,-80.131,441.572,172.568,22.526,154.088
C02572=1070.841,-80.381,441.583,172.566,22.525,154.088
C02573=1070.834,-80.631,441.593,172.565,22.523,154.088
C02574=1070.828,-80.880,441.604,172.563,22.521,154.088
C02575=1070.822,-81.130,441.615,172.562,22.520,154.088
C02576=1070.815,-81.380,441.626,172.560,22.519,154.088
C02577=1070.810,-81.621,441.636,172.559,22.517,154.088
C02578=1070.804,-81.862,441.647,172.557,22.516,154.088
C02579=1070.798,-82.103,441.657,172.555,22.514,154.088
C02580=1070.792,-82.344,441.668,172.554,22.512,154.087
C02581=1070.786,-82.585,441.678,172.552,22.511,154.087
C02582=1070.780,-82.826,441.689,172.551,22.510,154.087
C02583=1070.774,-83.068,441.698,172.549,22.508,154.087
C02584=1070.769,-83.309,441.709,172.548,22.506,154.087
C02585=1070.763,-83.559,441.720,172.546,22.505,154.087
C02586=1070.756,-83.809,441.730,172.545,22.504,154.087
C02587=1070.750,-84.058,441.741,172.543,22.502,154.087
C02588=1070.744,-84.308,441.752,172.542,22.500,154.087
C02589=1070.737,-84.558,441.763,172.540,22.499,154.087
C02590=1070.731,-84.807,441.774,172.539,22.497,154.087
C02591=1070.726,-85.057,441.785,172.537,22.496,154.087
C02592=1070.719,-85.307,441.795,172.535,22.494,154.087
C02593=1070.712,-85.604,441.807,172.533,22.492,154.087
C02594=1070.705,-85.900,441.820,172.531,22.491,154.087
C02595=1070.697,-86.198,441.833,172.529,22.488,154.087
C02596=1070.690,-86.495,441.845,172.527,22.487,154.087
C02597=1070.685,-86.744,441.856,172.526,22.486,154.087
C02598=1070.677,-86.994,441.867,172.524,22.484,154.086
C02599=1070.672,-87.243,441.878,172.523,22.482,154.086
C02600=1070.666,-87.493,441.887,172.521,22.481,154.086
C02601=1070.660,-87.743,441.898,172.520,22.480,154.086
C02602=1070.653,-87.993,441.909,172.518,22.478,154.086
C02603=1070.647,-88.242,441.920,172.517,22.476,154.086
C02604=1070.642,-88.492,441.930,172.515,22.475,154.086
C02605=1070.636,-88.742,441.941,172.513,22.474,154.086
C02606=1070.629,-88.992,441.951,172.512,22.472,154.086
C02607=1070.623,-89.241,441.962,172.510,22.470,154.086
C02608=1070.617,-89.491,441.972,172.509,22.469,154.086
C02609=1070.611,-89.740,441.983,172.507,22.468,154.086
C02610=1070.605,-89.991,441.994,172.506,22.466,154.086
C02611=1070.599,-90.240,442.004,172.504,22.465,154.086
C02612=1070.593,-90.490,442.014,172.503,22.463,154.086
C02613=1070.586,-90.739,442.025,172.501,22.462,154.086
C02614=1070.581,-90.989,442.036,172.499,22.460,154.086
C02615=1070.575,-91.239,442.046,172.498,22.459,154.086
C02616=1070.568,-91.489,442.056,172.496,22.458,154.086
C02617=1070.562,-91.738,442.067,172.495,22.456,154.086
C02618=1070.556,-91.988,442.077,172.493,22.455,154.086
C02619=1070.550,-92.237,442.088,172.492,22.453,154.086
C02620=1070.544,-92.487,442.099,172.490,22.452,154.086
C02621=1070.538,-92.737,442.108,172.488,22.450,154.085
C02622=1070.532,-92.987,442.119,172.487,22.449,154.085
C02623=1070.526,-93.237,442.129,172.485,22.448,154.085
C02624=1070.520,-93.486,442.140,172.484,22.446,154.085
C02625=1070.514,-93.735,442.150,172.482,22.445,154.085
C02626=1070.508,-93.986,442.161,172.480,22.444,154.085
C02627=1070.502,-94.236,442.171,172.479,22.442,154.085
C02628=1070.496,-94.485,442.181,172.477,22.440,154.085
C02629=1070.490,-94.735,442.192,172.476,22.439,154.085
C02630=1070.484,-94.984,442.202,172.474,22.438,154.085
C02631=1070.478,-95.234,442.212,172.472,22.436,154.085
C02632=1070.472,-95.483,442.223,172.471,22.435,154.085
C02633=1070.466,-95.733,442.233,172.469,22.434,154.085
C02634=1070.459,-95.983,442.243,172.468,22.432,154.085
C02635=1070.454,-96.233,442.254,172.466,22.431,154.085
C02636=1070.447,-96.483,442.264,172.464,22.429,154.085
C02637=1070.442,-96.733,442.274,172.463,22.428,154.085
C02638=1070.436,-96.982,442.285,172.461,22.427,154.085
C02639=1070.430,-97.232,442.295,172.460,22.425,154.085
C02640=1070.424,-97.481,442.305,172.458,22.424,154.085
C02641=1070.417,-97.763,442.316,172.456,22.423,154.085
C02642=1070.409,-98.046,442.329,172.454,22.421,154.085
C02643=1070.403,-98.328,442.340,172.452,22.420,154.085
C02644=1070.396,-98.610,442.351,172.451,22.418,154.085
C02645=1070.390,-98.860,442.361,172.449,22.417,154.085
C02646=1070.384,-99.110,442.372,172.448,22.416,154.085
C02647=1070.378,-99.360,442.382,172.446,22.414,154.085
C02648=1070.371,-99.609,442.392,172.444,22.413,154.085
C02649=1070.366,-99.859,442.402,172.443,22.411,154.085
C02650=1070.359,-100.109,442.412,172.441,22.410,154.085
C02651=1070.353,-100.358,442.422,172.440,22.409,154.085
C02652=1070.347,-100.608,442.433,172.438,22.407,154.085
C02653=1070.341,-100.858,442.442,172.436,22.407,154.085
C02654=1070.335,-101.107,442.452,172.435,22.405,154.085
C02655=1070.328,-101.357,442.462,172.433,22.404,154.085
C02656=1070.323,-101.607,442.472,172.431,22.403,154.085
C02657=1070.316,-101.857,442.483,172.430,22.401,154.085
C02658=1070.310,-102.106,442.493,172.428,22.400,154.085
C02659=1070.304,-102.357,442.503,172.426,22.399,154.085
C02660=1070.298,-102.606,442.513,172.425,22.398,154.085
C02661=1070.292,-102.856,442.523,172.423,22.396,154.085
C02662=1070.286,-103.106,442.533,172.422,22.395,154.085
C02663=1070.280,-103.355,442.543,172.420,22.394,154.085
C02664=1070.274,-103.605,442.553,172.418,22.393,154.085
C02665=1070.267,-103.854,442.562,172.417,22.391,154.085
C02666=1070.262,-104.104,442.573,172.415,22.390,154.085
C02667=1070.256,-104.354,442.583,172.413,22.389,154.085
C02668=1070.249,-104.603,442.592,172.412,22.388,154.085
C02669=1070.244,-104.853,442.603,172.410,22.387,154.085
C02670=1070.237,-105.103,442.613,172.408,22.385,154.085
C02671=1070.231,-105.353,442.622,172.407,22.384,154.085
C02672=1070.225,-105.602,442.632,172.405,22.383,154.085
C02673=1070.219,-105.852,442.643,172.403,22.382,154.085
C02674=1070.213,-106.102,442.652,172.403,22.381,154.085
C02675=1070.207,-106.351,442.662,172.401,22.379,154.085
C02676=1070.201,-106.601,442.671,172.399,22.379,154.085
C02677=1070.194,-106.851,442.682,172.398,22.377,154.085
C02678=1070.188,-107.101,442.692,172.396,22.376,154.085
C02679=1070.182,-107.351,442.702,172.394,22.375,154.085
C02680=1070.176,-107.601,442.711,172.393,22.374,154.085
C02681=1070.170,-107.850,442.722,172.391,22.372,154.085
C02682=1070.163,-108.100,442.731,172.389,22.372,154.085
C02683=1070.157,-108.350,442.741,172.388,22.370,154.085
C02684=1070.152,-108.600,442.751,172.386,22.369,154.085
C02685=1070.146,-108.850,442.760,172.384,22.368,154.086
C02686=1070.139,-109.099,442.771,172.383,22.367,154.086
C02687=1070.133,-109.349,442.780,172.381,22.366,154.086
C02688=1070.127,-109.598,442.790,172.379,22.365,154.086
C02689=1070.121,-109.848,442.799,172.378,22.364,154.086
C02690=1070.114,-110.098,442.809,172.376,22.362,154.086
C02691=1070.108,-110.348,442.818,172.374,22.361,154.086
C02692=1070.102,-110.597,442.828,172.373,22.360,154.086
C02693=1070.096,-110.847,442.838,172.371,22.359,154.086
C02694=1070.090,-111.097,442.848,172.369,22.358,154.086
C02695=1070.084,-111.347,442.858,172.368,22.357,154.086
C02696=1070.078,-111.596,442.868,172.366,22.356,154.086
C02697=1070.072,-111.846,442.877,172.364,22.355,154.086
C02698=1070.066,-112.095,442.886,172.362,22.354,154.086
C02699=1070.060,-112.345,442.896,172.362,22.353,154.086
C02700=1070.054,-112.595,442.906,172.360,22.352,154.086
C02701=1070.048,-112.845,442.915,172.358,22.351,154.086
C02702=1070.041,-113.094,442.925,172.357,22.349,154.086
C02703=1070.035,-113.344,442.935,172.355,22.349,154.086
C02704=1070.029,-113.593,442.945,172.353,22.347,154.086
C02705=1070.022,-113.873,442.955,172.352,22.346,154.086
C02706=1070.015,-114.154,442.966,172.349,22.345,154.086
C02707=1070.008,-114.434,442.976,172.347,22.344,154.087
C02708=1070.002,-114.713,442.987,172.346,22.342,154.086
C02709=1069.996,-114.963,442.997,172.344,22.342,154.087
C02710=1069.989,-115.213,443.006,172.342,22.341,154.087
C02711=1069.983,-115.463,443.016,172.340,22.339,154.087
C02712=1069.977,-115.713,443.025,172.339,22.339,154.087
C02713=1069.971,-115.962,443.035,172.337,22.337,154.087
C02714=1069.965,-116.212,443.045,172.335,22.337,154.087
C02715=1069.959,-116.462,443.054,172.333,22.336,154.087
C02716=1069.952,-116.712,443.064,172.333,22.335,154.087
C02717=1069.947,-116.961,443.073,172.331,22.334,154.087
C02718=1069.941,-117.211,443.082,172.329,22.333,154.087
C02719=1069.934,-117.461,443.092,172.328,22.332,154.087
C02720=1069.928,-117.710,443.102,172.326,22.331,154.087
C02721=1069.922,-117.960,443.111,172.324,22.330,154.087
C02722=1069.915,-118.210,443.120,172.322,22.329,154.087
C02723=1069.909,-118.459,443.130,172.321,22.328,154.088
C02724=1069.903,-118.709,443.139,172.319,22.327,154.088
C02725=1069.897,-118.959,443.149,172.317,22.326,154.088
C02726=1069.890,-119.209,443.158,172.315,22.325,154.088
C02727=1069.885,-119.459,443.167,172.314,22.324,154.088
C02728=1069.879,-119.708,443.176,172.312,22.323,154.088
C02729=1069.873,-119.958,443.186,172.310,22.322,154.088
C02730=1069.867,-120.208,443.196,172.309,22.321,154.088
C02731=1069.861,-120.458,443.205,172.308,22.320,154.088
C02732=1069.854,-120.707,443.214,172.306,22.320,154.088
C02733=1069.847,-120.957,443.224,172.304,22.319,154.088
C02734=1069.842,-121.206,443.233,172.302,22.318,154.088
C02735=1069.836,-121.457,443.242,172.301,22.317,154.088
C02736=1069.830,-121.706,443.251,172.299,22.316,154.088
C02737=1069.824,-121.956,443.261,172.297,22.315,154.089
C02738=1069.817,-122.206,443.270,172.295,22.314,154.089
C02739=1069.811,-122.455,443.279,172.294,22.313,154.089
C02740=1069.805,-122.706,443.288,172.292,22.312,154.089
C02741=1069.799,-122.955,443.297,172.290,22.311,154.089
C02742=1069.793,-123.205,443.307,172.289,22.311,154.089
C02743=1069.787,-123.455,443.317,172.287,22.310,154.089
C02744=1069.781,-123.704,443.326,172.286,22.309,154.089
C02745=1069.774,-123.954,443.334,172.284,22.308,154.089
C02746=1069.768,-124.203,443.344,172.282,22.307,154.089
C02747=1069.762,-124.453,443.353,172.281,22.306,154.089
C02748=1069.756,-124.703,443.363,172.279,22.306,154.090
C02749=1069.750,-124.954,443.372,172.277,22.305,154.090
C02750=1069.743,-125.203,443.381,172.275,22.304,154.090
C02751=1069.737,-125.453,443.390,172.274,22.303,154.090
C02752=1069.732,-125.702,443.399,172.272,22.302,154.090
C02753=1069.725,-125.952,443.408,172.270,22.302,154.090
C02754=1069.719,-126.202,443.417,172.268,22.300,154.090
C02755=1069.713,-126.452,443.427,172.267,22.300,154.090
C02756=1069.707,-126.702,443.436,172.266,22.299,154.090
C02757=1069.700,-126.951,443.444,172.264,22.298,154.090
C02758=1069.694,-127.201,443.454,172.262,22.297,154.091
C02759=1069.688,-127.450,443.463,172.260,22.297,154.091
C02760=1069.682,-127.701,443.472,172.259,22.296,154.091
C02761=1069.676,-127.951,443.481,172.257,22.295,154.091
C02762=1069.672,-128.202,443.491,172.255,22.294,154.091
C02763=1069.669,-128.453,443.501,172.254,22.291,154.091
C02764=1069.669,-128.703,443.513,172.253,22.289,154.090
C02765=1069.671,-128.956,443.526,172.252,22.285,154.090
C02766=1069.674,-129.209,443.539,172.251,22.280,154.089
C02767=1069.679,-129.460,443.554,172.252,22.276,154.088
C02768=1069.687,-129.711,443.568,172.252,22.270,154.087
C02769=1069.297,-129.732,443.400,172.205,22.411,154.119
C02770=1069.290,-129.482,443.386,172.205,22.417,154.121
C02771=1069.285,-129.231,443.371,172.205,22.422,154.121
C02772=1069.281,-128.979,443.358,172.206,22.427,154.122
C02773=1069.279,-128.725,443.345,172.207,22.430,154.123
C02774=1069.279,-128.475,443.334,172.208,22.434,154.123
C02775=1069.281,-128.224,443.323,172.208,22.435,154.123
C02776=1069.286,-127.973,443.313,172.210,22.437,154.123
C02777=1069.292,-127.723,443.304,172.211,22.438,154.123
C02778=1069.298,-127.473,443.294,172.213,22.439,154.123
C02779=1069.305,-127.224,443.285,172.215,22.439,154.123
C02780=1069.311,-126.973,443.276,172.217,22.440,154.123
C02781=1069.317,-126.723,443.267,172.219,22.441,154.123
C02782=1069.322,-126.474,443.258,172.220,22.442,154.123
C02783=1069.329,-126.225,443.249,172.222,22.442,154.123
C02784=1069.335,-125.974,443.240,172.224,22.443,154.122
C02785=1069.341,-125.724,443.230,172.226,22.444,154.122
C02786=1069.348,-125.475,443.221,172.227,22.445,154.122
C02787=1069.353,-125.225,443.213,172.228,22.445,154.122
C02788=1069.360,-124.976,443.203,172.230,22.447,154.122
C02789=1069.366,-124.726,443.194,172.232,22.447,154.122
C02790=1069.373,-124.476,443.185,172.234,22.448,154.122
C02791=1069.378,-124.226,443.176,172.235,22.449,154.122
C02792=1069.384,-123.977,443.167,172.237,22.450,154.122
C02793=1069.390,-123.727,443.157,172.239,22.451,154.122
C02794=1069.396,-123.477,443.148,172.241,22.451,154.121
C02795=1069.402,-123.227,443.139,172.242,22.453,154.121
C02796=1069.409,-122.977,443.130,172.244,22.453,154.121
C02797=1069.415,-122.727,443.120,172.246,22.454,154.121
C02798=1069.421,-122.478,443.111,172.248,22.455,154.121
C02799=1069.427,-122.229,443.101,172.250,22.456,154.121
C02800=1069.433,-121.979,443.092,172.250,22.457,154.121
C02801=1069.439,-121.728,443.083,172.252,22.458,154.121
C02802=1069.446,-121.479,443.074,172.254,22.458,154.121
C02803=1069.452,-121.229,443.064,172.256,22.459,154.121
C02804=1069.458,-120.979,443.055,172.257,22.461,154.121
C02805=1069.464,-120.730,443.046,172.259,22.461,154.121
C02806=1069.470,-120.480,443.036,172.261,22.462,154.121
C02807=1069.476,-120.230,443.027,172.263,22.463,154.120
C02808=1069.482,-119.980,443.018,172.264,22.464,154.120
C02809=1069.488,-119.730,443.008,172.266,22.465,154.120
C02810=1069.495,-119.481,442.999,172.268,22.466,154.120
C02811=1069.501,-119.231,442.990,172.269,22.467,154.120
C02812=1069.507,-118.982,442.980,172.271,22.468,154.120
C02813=1069.513,-118.732,442.971,172.273,22.469,154.120
C02814=1069.519,-118.482,442.961,172.274,22.470,154.120
C02815=1069.526,-118.233,442.952,172.275,22.470,154.120
C02816=1069.532,-117.983,442.942,172.277,22.471,154.120
C02817=1069.538,-117.733,442.933,172.279,22.473,154.120
C02818=1069.544,-117.483,442.924,172.281,22.473,154.120
C02819=1069.550,-117.233,442.914,172.282,22.474,154.120
C02820=1069.556,-116.983,442.905,172.284,22.476,154.120
C02821=1069.562,-116.733,442.895,172.286,22.476,154.119
C02822=1069.568,-116.484,442.886,172.288,22.477,154.119
C02823=1069.574,-116.234,442.876,172.289,22.478,154.119
C02824=1069.580,-115.984,442.867,172.291,22.479,154.119
C02825=1069.586,-115.735,442.857,172.293,22.481,154.119
C02826=1069.592,-115.485,442.847,172.294,22.481,154.119
C02827=1069.599,-115.235,442.839,172.296,22.482,154.119
C02828=1069.606,-114.986,442.829,172.298,22.484,154.119
C02829=1069.612,-114.736,442.819,172.300,22.484,154.119
C02830=1069.618,-114.456,442.809,172.301,22.486,154.119
C02831=1069.625,-114.175,442.798,172.303,22.486,154.119
C02832=1069.632,-113.896,442.786,172.305,22.488,154.119
C02833=1069.639,-113.616,442.776,172.306,22.489,154.119
C02834=1069.645,-113.367,442.767,172.308,22.490,154.119
C02835=1069.651,-113.116,442.756,172.310,22.491,154.119
C02836=1069.657,-112.867,442.747,172.311,22.492,154.119
C02837=1069.663,-112.617,442.737,172.313,22.493,154.119
C02838=1069.669,-112.367,442.728,172.315,22.494,154.119
C02839=1069.675,-112.117,442.718,172.317,22.495,154.118
C02840=1069.682,-111.867,442.709,172.318,22.496,154.118
C02841=1069.688,-111.618,442.699,172.320,22.497,154.118
C02842=1069.694,-111.368,442.689,172.322,22.499,154.118
C02843=1069.700,-111.119,442.679,172.323,22.500,154.118
C02844=1069.707,-110.869,442.670,172.325,22.501,154.118
C02845=1069.713,-110.619,442.660,172.327,22.502,154.118
C02846=1069.719,-110.369,442.650,172.328,22.503,154.118
C02847=1069.724,-110.119,442.640,172.330,22.504,154.118
C02848=1069.730,-109.869,442.631,172.332,22.505,154.118
C02849=1069.737,-109.620,442.621,172.333,22.506,154.118
C02850=1069.743,-109.370,442.611,172.335,22.508,154.118
C02851=1069.749,-109.121,442.601,172.337,22.508,154.118
C02852=1069.755,-108.871,442.592,172.338,22.510,154.118
C02853=1069.762,-108.621,442.582,172.340,22.511,154.118
C02854=1069.768,-108.371,442.573,172.342,22.512,154.118
C02855=1069.774,-108.121,442.563,172.342,22.513,154.118
C02856=1069.780,-107.872,442.552,172.344,22.514,154.118
C02857=1069.786,-107.622,442.543,172.346,22.515,154.118
C02858=1069.792,-107.372,442.533,172.347,22.516,154.118
C02859=1069.798,-107.123,442.523,172.349,22.517,154.118
C02860=1069.805,-106.873,442.513,172.351,22.518,154.118
C02861=1069.810,-106.623,442.503,172.352,22.520,154.118
C02862=1069.816,-106.373,442.493,172.354,22.521,154.118
C02863=1069.822,-106.124,442.484,172.356,22.522,154.118
C02864=1069.829,-105.874,442.474,172.357,22.523,154.118
C02865=1069.835,-105.625,442.464,172.359,22.525,154.118
C02866=1069.841,-105.375,442.454,172.361,22.525,154.118
C02867=1069.847,-105.125,442.444,172.362,22.527,154.118
C02868=1069.853,-104.876,442.434,172.364,22.528,154.118
C02869=1069.859,-104.626,442.424,172.366,22.530,154.118
C02870=1069.865,-104.376,442.414,172.367,22.530,154.118
C02871=1069.871,-104.127,442.404,172.369,22.532,154.118
C02872=1069.877,-103.877,442.394,172.371,22.533,154.118
C02873=1069.884,-103.626,442.384,172.372,22.534,154.118
C02874=1069.890,-103.377,442.374,172.374,22.535,154.117
C02875=1069.896,-103.127,442.364,172.376,22.536,154.117
C02876=1069.902,-102.877,442.354,172.377,22.538,154.118
C02877=1069.908,-102.628,442.344,172.379,22.539,154.118
C02878=1069.914,-102.378,442.334,172.381,22.541,154.118
C02879=1069.920,-102.128,442.324,172.382,22.542,154.118
C02880=1069.926,-101.879,442.314,172.384,22.543,154.117
C02881=1069.932,-101.629,442.304,172.386,22.544,154.117
C02882=1069.939,-101.380,442.294,172.387,22.545,154.117
C02883=1069.944,-101.129,442.284,172.389,22.547,154.117
C02884=1069.950,-100.880,442.274,172.390,22.548,154.117
C02885=1069.957,-100.630,442.264,172.392,22.549,154.118
C02886=1069.963,-100.380,442.253,172.394,22.550,154.117
C02887=1069.969,-100.130,442.243,172.395,22.552,154.117
C02888=1069.976,-99.881,442.233,172.397,22.553,154.117
C02889=1069.982,-99.631,442.224,172.399,22.554,154.117
C02890=1069.987,-99.381,442.213,172.400,22.556,154.117
C02891=1069.994,-99.132,442.203,172.402,22.557,154.117
C02892=1069.999,-98.882,442.192,172.403,22.558,154.117
C02893=1070.006,-98.632,442.183,172.405,22.560,154.118
C02894=1070.013,-98.349,442.171,172.407,22.561,154.118
C02895=1070.020,-98.068,442.159,172.408,22.562,154.118
C02896=1070.027,-97.786,442.148,172.410,22.564,154.118
C02897=1070.034,-97.503,442.137,172.412,22.565,154.118
C02898=1070.040,-97.253,442.126,172.414,22.567,154.118
C02899=1070.046,-97.003,442.116,172.416,22.568,154.118
C02900=1070.052,-96.754,442.105,172.417,22.569,154.118
C02901=1070.058,-96.504,442.096,172.419,22.571,154.118
C02902=1070.064,-96.255,442.085,172.420,22.572,154.118
C02903=1070.070,-96.005,442.075,172.422,22.574,154.118
C02904=1070.076,-95.755,442.065,172.424,22.575,154.118
C02905=1070.082,-95.505,442.054,172.425,22.576,154.118
C02906=1070.088,-95.255,442.044,172.427,22.578,154.118
C02907=1070.094,-95.006,442.033,172.428,22.579,154.118
C02908=1070.100,-94.756,442.023,172.430,22.581,154.118
C02909=1070.106,-94.507,442.012,172.431,22.582,154.118
C02910=1070.112,-94.257,442.003,172.433,22.584,154.118
C02911=1070.118,-94.007,441.992,172.435,22.585,154.118
C02912=1070.125,-93.757,441.981,172.436,22.586,154.118
C02913=1070.130,-93.507,441.971,172.438,22.588,154.118
C02914=1070.136,-93.258,441.960,172.440,22.589,154.118
C02915=1070.142,-93.008,441.951,172.441,22.590,154.118
C02916=1070.148,-92.759,441.940,172.443,22.592,154.118
C02917=1070.154,-92.509,441.930,172.444,22.594,154.118
C02918=1070.160,-92.259,441.919,172.446,22.595,154.118
C02919=1070.167,-92.009,441.909,172.447,22.596,154.118
C02920=1070.173,-91.760,441.898,172.449,22.598,154.118
C02921=1070.178,-91.510,441.888,172.451,22.599,154.118
C02922=1070.184,-91.261,441.877,172.452,22.600,154.118
C02923=1070.191,-91.010,441.866,172.454,22.602,154.118
C02924=1070.197,-90.761,441.857,172.455,22.604,154.118
C02925=1070.203,-90.511,441.846,172.457,22.605,154.118
C02926=1070.208,-90.262,441.835,172.458,22.606,154.118
C02927=1070.215,-90.012,441.825,172.460,22.608,154.118
C02928=1070.221,-89.762,441.814,172.461,22.609,154.119
C02929=1070.227,-89.512,441.804,172.463,22.611,154.119
C02930=1070.233,-89.263,441.793,172.465,22.612,154.119
C02931=1070.239,-89.013,441.783,172.466,22.614,154.119
C02932=1070.246,-88.763,441.772,172.468,22.615,154.119
C02933=1070.251,-88.514,441.761,172.469,22.617,154.119
C02934=1070.257,-88.264,441.750,172.471,22.618,154.119
C02935=1070.263,-88.014,441.741,172.473,22.619,154.119
C02936=1070.270,-87.764,441.729,172.474,22.621,154.119
C02937=1070.276,-87.515,441.719,172.476,22.622,154.119
C02938=1070.282,-87.265,441.708,172.477,22.624,154.119
C02939=1070.288,-87.016,441.697,172.479,22.625,154.119
C02940=1070.294,-86.765,441.688,172.480,22.627,154.119
C02941=1070.300,-86.516,441.677,172.482,22.628,154.119
C02942=1070.306,-86.266,441.666,172.483,22.630,154.119
C02943=1070.313,-86.017,441.655,172.485,22.631,154.119
C02944=1070.319,-85.767,441.644,172.487,22.633,154.119
C02945=1070.324,-85.517,441.634,172.488,22.635,154.119
C02946=1070.331,-85.268,441.624,172.490,22.636,154.119
C02947=1070.337,-85.018,441.613,172.491,22.637,154.119
C02948=1070.343,-84.768,441.602,172.493,22.639,154.119
C02949=1070.349,-84.519,441.591,172.494,22.641,154.120
C02950=1070.356,-84.269,441.580,172.496,22.642,154.120
C02951=1070.361,-84.019,441.569,172.498,22.643,154.120
C02952=1070.368,-83.770,441.559,172.499,22.645,154.120
C02953=1070.374,-83.519,441.548,172.501,22.646,154.120
C02954=1070.380,-83.270,441.538,172.502,22.648,154.120
C02955=1070.386,-83.021,441.527,172.504,22.650,154.120
C02956=1070.392,-82.770,441.516,172.505,22.651,154.120
C02957=1070.398,-82.521,441.505,172.507,22.652,154.120
C02958=1070.405,-82.241,441.493,172.509,22.655,154.120
C02959=1070.412,-81.961,441.481,172.511,22.656,154.120
C02960=1070.419,-81.681,441.469,172.512,22.658,154.120
C02961=1070.426,-81.400,441.457,172.514,22.659,154.120
C02962=1070.432,-81.151,441.447,172.515,22.661,154.120
C02963=1070.438,-80.902,441.436,172.518,22.663,154.120
C02964=1070.444,-80.651,441.424,172.519,22.664,154.120
C02965=1070.451,-80.402,441.414,172.521,22.666,154.120
C02966=1070.457,-80.152,441.403,172.522,22.668,154.120
C02967=1070.463,-79.903,441.392,172.524,22.669,154.121
C02968=1070.469,-79.653,441.381,172.525,22.671,154.121
C02969=1070.475,-79.403,441.370,172.527,22.673,154.121
C02970=1070.481,-79.153,441.359,172.529,22.674,154.121
C02971=1070.487,-78.904,441.349,172.530,22.676,154.121
C02972=1070.494,-78.654,441.337,172.532,22.677,154.121
C02973=1070.499,-78.405,441.327,172.533,22.679,154.121
C02974=1070.505,-78.155,441.316,172.535,22.681,154.121
C02975=1070.511,-77.905,441.304,172.536,22.682,154.121
C02976=1070.518,-77.656,441.293,172.538,22.684,154.121
C02977=1070.524,-77.406,441.282,172.539,22.686,154.121
C02978=1070.530,-77.156,441.271,172.541,22.687,154.121
C02979=1070.535,-76.907,441.260,172.542,22.689,154.122
C02980=1070.542,-76.657,441.249,172.544,22.690,154.122
C02981=1070.548,-76.407,441.238,172.545,22.692,154.122
C02982=1070.554,-76.158,441.227,172.547,22.694,154.122
C02983=1070.560,-75.908,441.216,172.548,22.695,154.122
C02984=1070.566,-75.658,441.205,172.550,22.697,154.122
C02985=1070.572,-75.408,441.194,172.551,22.699,154.122
C02986=1070.578,-75.159,441.183,172.553,22.701,154.122
C02987=1070.585,-74.909,441.171,172.554,22.702,154.122
C02988=1070.590,-74.660,441.160,172.556,22.704,154.122
C02989=1070.596,-74.410,441.150,172.557,22.706,154.123
C02990=1070.603,-74.160,441.138,172.559,22.707,154.123
C02991=1070.608,-73.910,441.127,172.561,22.709,154.123
C02992=1070.615,-73.661,441.115,172.563,22.711,154.123
C02993=1070.621,-73.411,441.105,172.564,22.713,154.123
C02994=1070.626,-73.162,441.094,172.566,22.715,154.123
C02995=1070.633,-72.912,441.082,172.567,22.716,154.123
C02996=1070.638,-72.662,441.071,172.569,22.718,154.123
C02997=1070.644,-72.412,441.059,172.570,22.720,154.123
C02998=1070.650,-72.163,441.048,172.571,22.722,154.123
C02999=1070.656,-71.913,441.037,172.573,22.723,154.124
C03000=1070.662,-71.663,441.026,172.575,22.725,154.124
C03001=1070.668,-71.414,441.015,172.576,22.727,154.124
C03002=1070.675,-71.164,441.003,172.577,22.729,154.124
C03003=1070.680,-70.914,440.992,172.579,22.731,154.124
C03004=1070.685,-70.665,440.981,172.580,22.732,154.124
C03005=1070.692,-70.415,440.969,172.582,22.734,154.124
C03006=1070.698,-70.166,440.958,172.583,22.736,154.124
C03007=1070.704,-69.915,440.947,172.585,22.738,154.125
C03008=1070.710,-69.666,440.936,172.586,22.739,154.125
C03009=1070.716,-69.416,440.923,172.588,22.741,154.125
C03010=1070.721,-69.167,440.912,172.589,22.743,154.125
C03011=1070.727,-68.917,440.902,172.591,22.745,154.125
C03012=1070.734,-68.668,440.890,172.593,22.747,154.125
C03013=1070.740,-68.418,440.879,172.594,22.749,154.125
C03014=1070.745,-68.168,440.867,172.596,22.750,154.125
C03015=1070.751,-67.919,440.855,172.597,22.752,154.125
C03016=1070.758,-67.668,440.844,172.599,22.754,154.126
C03017=1070.763,-67.419,440.833,172.600,22.756,154.126
C03018=1070.770,-67.169,440.821,172.602,22.758,154.126
C03019=1070.775,-66.920,440.810,172.603,22.760,154.126
C03020=1070.782,-66.670,440.798,172.605,22.761,154.126
C03021=1070.787,-66.421,440.787,172.606,22.763,154.126
C03022=1070.795,-66.143,440.774,172.608,22.765,154.126
C03023=1070.801,-65.865,440.761,172.610,22.767,154.126
C03024=1070.807,-65.587,440.749,172.611,22.769,154.127
C03025=1070.814,-65.309,440.736,172.613,22.771,154.127
C03026=1070.820,-65.060,440.724,172.614,22.773,154.127
C03027=1070.826,-64.810,440.713,172.616,22.775,154.127
C03028=1070.833,-64.560,440.701,172.617,22.777,154.127
C03029=1070.838,-64.310,440.689,172.619,22.778,154.127
C03030=1070.844,-64.061,440.678,172.620,22.780,154.127
C03031=1070.850,-63.811,440.667,172.622,22.783,154.128
C03032=1070.857,-63.562,440.655,172.624,22.785,154.128
C03033=1070.863,-63.312,440.644,172.625,22.786,154.128
C03034=1070.868,-63.062,440.631,172.627,22.788,154.128
C03035=1070.874,-62.813,440.620,172.628,22.790,154.128
C03036=1070.881,-62.563,440.608,172.630,22.792,154.128
C03037=1070.887,-62.314,440.598,172.631,22.793,154.128
C03038=1070.892,-62.064,440.585,172.633,22.795,154.128
C03039=1070.899,-61.814,440.574,172.634,22.797,154.129
C03040=1070.905,-61.565,440.562,172.635,22.799,154.129
C03041=1070.910,-61.314,440.550,172.637,22.801,154.129
C03042=1070.917,-61.065,440.539,172.638,22.803,154.129
C03043=1070.923,-60.815,440.527,172.640,22.805,154.129
C03044=1070.929,-60.566,440.516,172.641,22.807,154.129
C03045=1070.934,-60.316,440.504,172.643,22.809,154.130
C03046=1070.941,-60.066,440.492,172.644,22.811,154.130
C03047=1070.947,-59.817,440.481,172.647,22.812,154.130
C03048=1070.953,-59.567,440.469,172.648,22.814,154.130
C03049=1070.959,-59.317,440.457,172.649,22.816,154.130
C03050=1070.965,-59.068,440.446,172.651,22.818,154.130
C03051=1070.972,-58.818,440.434,172.652,22.820,154.130
C03052=1070.978,-58.568,440.421,172.654,22.822,154.130
C03053=1070.983,-58.319,440.410,172.655,22.824,154.131
C03054=1070.990,-58.069,440.398,172.657,22.826,154.131
C03055=1070.996,-57.819,440.387,172.658,22.827,154.131
C03056=1071.002,-57.570,440.375,172.660,22.829,154.131
C03057=1071.008,-57.320,440.363,172.661,22.831,154.131
C03058=1071.014,-57.070,440.351,172.662,22.833,154.131
C03059=1071.020,-56.821,440.340,172.664,22.835,154.131
C03060=1071.027,-56.571,440.328,172.665,22.837,154.132
C03061=1071.032,-56.321,440.316,172.667,22.839,154.132
C03062=1071.038,-56.072,440.304,172.669,22.841,154.132
C03063=1071.045,-55.822,440.292,172.671,22.843,154.132
C03064=1071.051,-55.572,440.280,172.672,22.845,154.132
C03065=1071.057,-55.323,440.269,172.673,22.847,154.132
C03066=1071.063,-55.073,440.257,172.675,22.849,154.132
C03067=1071.069,-54.824,440.244,172.676,22.851,154.133
C03068=1071.075,-54.574,440.233,172.678,22.852,154.133
C03069=1071.082,-54.324,440.222,172.679,22.854,154.133
C03070=1071.087,-54.075,440.209,172.681,22.856,154.133
C03071=1071.094,-53.825,440.197,172.682,22.858,154.133
C03072=1071.100,-53.576,440.186,172.683,22.860,154.133
C03073=1071.106,-53.326,440.174,172.685,22.862,154.133
C03074=1071.112,-53.076,440.162,172.686,22.864,154.134
C03075=1071.119,-52.827,440.150,172.688,22.866,154.134
C03076=1071.124,-52.577,440.137,172.690,22.869,154.134
C03077=1071.131,-52.327,440.126,172.691,22.870,154.134
C03078=1071.137,-52.078,440.114,172.693,22.872,154.134
C03079=1071.143,-51.828,440.102,172.694,22.874,154.134
C03080=1071.149,-51.579,440.090,172.696,22.876,154.135
C03081=1071.155,-51.329,440.078,172.697,22.878,154.135
C03082=1071.162,-51.097,440.067,172.699,22.880,154.135
C03083=1071.167,-50.864,440.055,172.700,22.882,154.135
C03084=1071.172,-50.633,440.044,172.701,22.884,154.135
C03085=1071.179,-50.400,440.034,172.703,22.886,154.135
C03086=1071.184,-50.168,440.022,172.704,22.887,154.135
C03087=1071.190,-49.937,440.011,172.705,22.889,154.136
C03088=1071.195,-49.704,439.999,172.706,22.891,154.136
C03089=1071.204,-49.348,439.982,172.708,22.894,154.136
C03090=1071.213,-48.974,439.963,172.711,22.897,154.136
C03091=1071.219,-48.724,439.952,172.713,22.899,154.136
C03092=1071.224,-48.475,439.940,172.714,22.901,154.137
C03093=1071.230,-48.225,439.927,172.716,22.903,154.137
C03094=1071.237,-47.976,439.915,172.717,22.905,154.137
C03095=1071.242,-47.726,439.903,172.718,22.908,154.137
C03096=1071.248,-47.477,439.891,172.720,22.909,154.137
C03097=1071.255,-47.227,439.879,172.721,22.911,154.138
C03098=1071.261,-46.977,439.866,172.723,22.914,154.138
C03099=1071.266,-46.728,439.854,172.724,22.916,154.138
C03100=1071.272,-46.478,439.842,172.725,22.918,154.138
C03101=1071.278,-46.228,439.829,172.727,22.919,154.138
C03102=1071.284,-45.979,439.817,172.728,22.922,154.139
C03103=1071.291,-45.729,439.805,172.730,22.924,154.139
C03104=1071.296,-45.480,439.793,172.732,22.926,154.139
C03105=1071.302,-45.230,439.780,172.733,22.928,154.139
C03106=1071.309,-44.980,439.768,172.735,22.930,154.139
C03107=1071.315,-44.731,439.756,172.736,22.932,154.139
C03108=1071.320,-44.481,439.743,172.737,22.935,154.140
C03109=1071.327,-44.232,439.732,172.739,22.937,154.140
C03110=1071.333,-43.982,439.719,172.740,22.938,154.140
C03111=1071.338,-43.732,439.706,172.742,22.940,154.140
C03112=1071.344,-43.482,439.694,172.743,22.943,154.140
C03113=1071.350,-43.233,439.682,172.744,22.945,154.141
C03114=1071.356,-42.983,439.670,172.746,22.947,154.141
C03115=1071.363,-42.734,439.656,172.747,22.949,154.141
C03116=1071.369,-42.485,439.644,172.749,22.951,154.141
C03117=1071.375,-42.235,439.632,172.751,22.953,154.141
C03118=1071.381,-41.985,439.619,172.752,22.956,154.141
C03119=1071.386,-41.736,439.607,172.754,22.958,154.142
C03120=1071.393,-41.486,439.595,172.755,22.959,154.142
C03121=1071.399,-41.236,439.583,172.756,22.962,154.142
C03122=1071.405,-40.986,439.570,172.758,22.964,154.142
C03123=1071.411,-40.737,439.557,172.759,22.966,154.142
C03124=1071.418,-40.487,439.545,172.760,22.968,154.143
C03125=1071.424,-40.238,439.532,172.762,22.970,154.143
C03126=1071.429,-39.988,439.520,172.763,22.972,154.143
C03127=1071.435,-39.738,439.508,172.765,22.974,154.143
C03128=1071.441,-39.489,439.496,172.767,22.977,154.143
C03129=1071.448,-39.240,439.482,172.768,22.979,154.144
C03130=1071.454,-38.990,439.470,172.770,22.981,154.144
C03131=1071.459,-38.740,439.457,172.771,22.983,154.144
C03132=1071.466,-38.490,439.445,172.772,22.985,154.144
C03133=1071.472,-38.240,439.433,172.774,22.987,154.144
C03134=1071.478,-37.991,439.419,172.775,22.990,154.145
C03135=1071.484,-37.742,439.407,172.777,22.991,154.145
C03136=1071.489,-37.492,439.395,172.778,22.994,154.145
C03137=1071.495,-37.242,439.382,172.779,22.996,154.145
C03138=1071.502,-36.993,439.369,172.780,22.998,154.145
C03139=1071.507,-36.743,439.356,172.783,23.000,154.146
C03140=1071.513,-36.493,439.344,172.784,23.003,154.146
C03141=1071.519,-36.243,439.331,172.786,23.005,154.146
C03142=1071.525,-35.994,439.318,172.787,23.007,154.146
C03143=1071.531,-35.745,439.306,172.788,23.009,154.146
C03144=1071.537,-35.495,439.293,172.790,23.012,154.147
C03145=1071.543,-35.246,439.280,172.791,23.013,154.147
C03146=1071.549,-34.996,439.267,172.792,23.016,154.147
C03147=1071.555,-34.746,439.255,172.794,23.018,154.147
C03148=1071.561,-34.497,439.242,172.795,23.020,154.148
C03149=1071.567,-34.247,439.229,172.796,23.022,154.148
C03150=1071.574,-33.971,439.215,172.799,23.025,154.148
C03151=1071.580,-33.695,439.201,172.800,23.027,154.148
C03152=1071.587,-33.419,439.186,172.801,23.030,154.149
C03153=1071.594,-33.143,439.173,172.803,23.033,154.149
C03154=1071.600,-32.893,439.160,172.805,23.035,154.149
C03155=1071.606,-32.643,439.147,172.806,23.037,154.149
C03156=1071.612,-32.394,439.135,172.807,23.039,154.149
C03157=1071.618,-32.144,439.122,172.809,23.041,154.150
C03158=1071.624,-31.895,439.109,172.810,23.043,154.150
C03159=1071.630,-31.645,439.096,172.811,23.046,154.150
C03160=1071.636,-31.395,439.084,172.813,23.048,154.150
C03161=1071.642,-31.146,439.070,172.814,23.050,154.150
C03162=1071.647,-30.896,439.057,172.815,23.052,154.151
C03163=1071.653,-30.647,439.044,172.818,23.055,154.151
C03164=1071.659,-30.397,439.031,172.819,23.057,154.151
C03165=1071.665,-30.147,439.018,172.821,23.059,154.151
C03166=1071.671,-29.898,439.006,172.822,23.061,154.152
C03167=1071.677,-29.648,438.992,172.823,23.063,154.152
C03168=1071.683,-29.398,438.980,172.825,23.066,154.152
C03169=1071.690,-29.149,438.966,172.826,23.068,154.152
C03170=1071.695,-28.899,438.954,172.827,23.070,154.152
C03171=1071.702,-28.650,438.941,172.829,23.072,154.153
C03172=1071.708,-28.400,438.928,172.830,23.074,154.153
C03173=1071.714,-28.151,438.915,172.831,23.077,154.153
C03174=1071.720,-27.901,438.902,172.834,23.079,154.153
C03175=1071.726,-27.652,438.889,172.835,23.082,154.154
C03176=1071.732,-27.402,438.876,172.836,23.084,154.154
C03177=1071.739,-27.152,438.863,172.838,23.086,154.154
C03178=1071.745,-26.902,438.850,172.839,23.088,154.154
C03179=1071.751,-26.653,438.837,172.840,23.090,154.154
C03180=1071.757,-26.403,438.824,172.842,23.093,154.155
C03181=1071.762,-26.153,438.811,172.843,23.095,154.155
C03182=1071.768,-25.904,438.797,172.844,23.097,154.155
C03183=1071.774,-25.654,438.785,172.846,23.099,154.155
C03184=1071.780,-25.405,438.771,172.847,23.102,154.156
C03185=1071.786,-25.155,438.758,172.849,23.105,154.156
C03186=1071.792,-24.905,438.745,172.851,23.106,154.156
C03187=1071.798,-24.656,438.732,172.852,23.109,154.156
C03188=1071.804,-24.406,438.719,172.853,23.111,154.157
C03189=1071.809,-24.157,438.705,172.855,23.113,154.157
C03190=1071.816,-23.907,438.692,172.856,23.116,154.157
C03191=1071.822,-23.658,438.680,172.857,23.118,154.157
C03192=1071.828,-23.408,438.666,172.858,23.121,154.158
C03193=1071.833,-23.159,438.652,172.860,23.122,154.158
C03194=1071.839,-22.909,438.640,172.861,23.125,154.158
C03195=1071.845,-22.660,438.627,172.863,23.128,154.158
C03196=1071.851,-22.410,438.613,172.865,23.130,154.159
C03197=1071.857,-22.160,438.600,172.866,23.132,154.159
C03198=1071.863,-21.911,438.587,172.867,23.134,154.159
C03199=1071.869,-21.662,438.574,172.869,23.137,154.159
C03200=1071.875,-21.412,438.560,172.870,23.139,154.159
C03201=1071.881,-21.162,438.547,172.871,23.141,154.160
C03202=1071.887,-20.912,438.534,172.873,23.144,154.160
C03203=1071.893,-20.663,438.520,172.874,23.146,154.160
C03204=1071.899,-20.413,438.506,172.875,23.148,154.160
C03205=1071.905,-20.163,438.494,172.877,23.150,154.161
C03206=1071.911,-19.914,438.481,172.879,23.153,154.161
C03207=1071.917,-19.665,438.467,172.880,23.156,154.161
C03208=1071.923,-19.415,438.453,172.882,23.157,154.161
C03209=1071.929,-19.166,438.440,172.883,23.160,154.162
C03210=1071.934,-18.916,438.427,172.884,23.162,154.162
C03211=1071.941,-18.666,438.413,172.885,23.165,154.162
C03212=1071.947,-18.417,438.400,172.887,23.167,154.162
C03213=1071.953,-18.167,438.386,172.888,23.169,154.163
C03214=1071.959,-17.891,438.372,172.890,23.172,154.163
C03215=1071.967,-17.614,438.357,172.892,23.174,154.163
C03216=1071.973,-17.336,438.341,172.893,23.177,154.163
C03217=1071.980,-17.060,438.327,172.895,23.180,154.164
C03218=1071.986,-16.810,438.314,172.896,23.182,154.164
C03219=1071.992,-16.560,438.300,172.898,23.184,154.164
C03220=1071.998,-16.310,438.287,172.899,23.187,154.165
C03221=1072.004,-16.061,438.274,172.900,23.189,154.165
C03222=1072.010,-15.812,438.260,172.902,23.191,154.165
C03223=1072.016,-15.562,438.246,172.903,23.194,154.165
C03224=1072.022,-15.313,438.233,172.904,23.196,154.166
C03225=1072.028,-15.063,438.219,172.905,23.198,154.166
C03226=1072.034,-14.814,438.206,172.907,23.200,154.166
C03227=1072.040,-14.564,438.192,172.909,23.203,154.166
C03228=1072.046,-14.314,438.179,172.910,23.206,154.166
C03229=1072.051,-14.064,438.165,172.912,23.208,154.167
C03230=1072.057,-13.815,438.152,172.913,23.210,154.167
C03231=1072.064,-13.565,438.138,172.914,23.213,154.167
C03232=1072.069,-13.315,438.124,172.916,23.215,154.168
C03233=1072.075,-13.066,438.111,172.917,23.218,154.168
C03234=1072.081,-12.817,438.097,172.918,23.220,154.168
C03235=1072.087,-12.567,438.084,172.920,23.222,154.168
C03236=1072.092,-12.318,438.070,172.921,23.224,154.169
C03237=1072.099,-12.068,438.056,172.923,23.227,154.169
C03238=1072.105,-11.818,438.042,172.924,23.230,154.169
C03239=1072.111,-11.569,438.029,172.926,23.232,154.169
C03240=1072.116,-11.319,438.015,172.927,23.234,154.170
C03241=1072.123,-11.070,438.002,172.928,23.237,154.170
C03242=1072.129,-10.820,437.988,172.929,23.239,154.170
C03243=1072.134,-10.571,437.973,172.931,23.242,154.171
C03244=1072.141,-10.322,437.960,172.932,23.244,154.171
C03245=1072.146,-10.072,437.946,172.934,23.246,154.171
C03246=1072.153,-9.822,437.932,172.935,23.248,154.171
C03247=1072.158,-9.572,437.918,172.937,23.251,154.171
C03248=1072.165,-9.323,437.905,172.938,23.254,154.172
C03249=1072.170,-9.074,437.891,172.940,23.256,154.172
C03250=1072.176,-8.823,437.877,172.941,23.259,154.172
C03251=1072.182,-8.574,437.864,172.942,23.261,154.173
C03252=1072.188,-8.324,437.850,172.943,23.263,154.173
C03253=1072.194,-8.076,437.836,172.945,23.266,154.173
C03254=1072.200,-7.826,437.822,172.946,23.268,154.173
C03255=1072.206,-7.576,437.808,172.947,23.270,154.174
C03256=1072.212,-7.327,437.795,172.949,23.273,154.174
C03257=1072.218,-7.077,437.781,172.951,23.275,154.174
C03258=1072.224,-6.827,437.767,172.952,23.278,154.174
C03259=1072.230,-6.578,437.752,172.954,23.280,154.175
C03260=1072.236,-6.329,437.739,172.955,23.283,154.175
C03261=1072.243,-6.079,437.725,172.956,23.285,154.175
C03262=1072.248,-5.829,437.711,172.957,23.287,154.176
C03263=1072.253,-5.580,437.697,172.959,23.290,154.176
C03264=1072.260,-5.331,437.683,172.960,23.292,154.176
C03265=1072.266,-5.081,437.669,172.961,23.295,154.176
C03266=1072.272,-4.831,437.656,172.963,23.297,154.177
C03267=1072.278,-4.582,437.642,172.965,23.299,154.177
C03268=1072.284,-4.331,437.628,172.966,23.302,154.177
C03269=1072.290,-4.083,437.614,172.968,23.304,154.177
C03270=1072.296,-3.833,437.600,172.969,23.307,154.178
C03271=1072.302,-3.583,437.586,172.970,23.309,154.178
C03272=1072.308,-3.334,437.572,172.971,23.312,154.178
C03273=1072.314,-3.085,437.558,172.973,23.314,154.178
C03274=1072.320,-2.834,437.543,172.974,23.316,154.179
C03275=1072.325,-2.585,437.530,172.975,23.319,154.179
C03276=1072.331,-2.336,437.515,172.977,23.322,154.179
C03277=1072.337,-2.086,437.501,172.979,23.324,154.180
C03278=1072.344,-1.808,437.485,172.980,23.327,154.180
C03279=1072.350,-1.529,437.470,172.981,23.329,154.180
C03280=1072.357,-1.251,437.454,172.983,23.333,154.181
C03281=1072.363,-0.972,437.438,172.984,23.335,154.181
C03282=1072.369,-0.722,437.424,172.986,23.338,154.181
C03283=1072.376,-0.473,437.410,172.987,23.340,154.181
C03284=1072.381,-0.224,437.396,172.988,23.342,154.182
C03285=1072.387,0.026,437.381,172.990,23.345,154.182
C03286=1072.393,0.276,437.367,172.992,23.348,154.182
C03287=1072.398,0.525,437.353,172.993,23.351,154.183
C03288=1072.405,0.775,437.338,172.994,23.353,154.183
C03289=1072.410,1.024,437.324,172.996,23.355,154.183
C03290=1072.416,1.273,437.310,172.997,23.358,154.183
C03291=1072.422,1.524,437.296,172.998,23.360,154.184
C03292=1072.428,1.773,437.281,172.999,23.363,154.184
C03293=1072.433,2.022,437.267,173.001,23.365,154.184
C03294=1072.439,2.273,437.253,173.002,23.368,154.185
C03295=1072.446,2.521,437.239,173.003,23.370,154.185
C03296=1072.452,2.771,437.225,173.006,23.373,154.185
C03297=1072.458,3.020,437.210,173.007,23.375,154.185
C03298=1072.463,3.270,437.196,173.008,23.378,154.186
C03299=1072.470,3.520,437.181,173.009,23.380,154.186
C03300=1072.475,3.769,437.168,173.011,23.383,154.186
C03301=1072.481,4.018,437.153,173.012,23.385,154.187
C03302=1072.487,4.268,437.139,173.013,23.388,154.187
C03303=1072.493,4.517,437.124,173.014,23.390,154.187
C03304=1072.499,4.768,437.110,173.016,23.393,154.188
C03305=1072.505,5.017,437.095,173.018,23.395,154.188
C03306=1072.510,5.266,437.081,173.019,23.398,154.188
C03307=1072.516,5.516,437.067,173.021,23.400,154.188
C03308=1072.522,5.765,437.052,173.022,23.403,154.189
C03309=1072.528,6.015,437.038,173.023,23.405,154.189
C03310=1072.534,6.264,437.023,173.024,23.408,154.189
C03311=1072.540,6.514,437.009,173.026,23.410,154.189
C03312=1072.546,6.763,436.994,173.027,23.412,154.190
C03313=1072.552,7.014,436.980,173.028,23.415,154.190
C03314=1072.558,7.263,436.966,173.030,23.418,154.190
C03315=1072.564,7.511,436.951,173.032,23.421,154.191
C03316=1072.570,7.762,436.937,173.033,23.423,154.191
C03317=1072.575,8.011,436.922,173.034,23.425,154.191
C03318=1072.582,8.260,436.907,173.036,23.428,154.192
C03319=1072.587,8.510,436.893,173.037,23.430,154.192
C03320=1072.594,8.760,436.878,173.038,23.433,154.192
C03321=1072.600,9.009,436.864,173.039,23.435,154.192
C03322=1072.606,9.259,436.850,173.041,23.437,154.193
C03323=1072.611,9.508,436.835,173.042,23.440,154.193
C03324=1072.618,9.757,436.820,173.044,23.443,154.193
C03325=1072.623,10.007,436.806,173.046,23.445,154.193
C03326=1072.630,10.257,436.791,173.047,23.448,154.194
C03327=1072.635,10.506,436.777,173.048,23.450,154.194
C03328=1072.641,10.756,436.762,173.049,23.453,154.194
C03329=1072.647,11.005,436.748,173.051,23.455,154.195
C03330=1072.654,11.255,436.733,173.052,23.458,154.195
C03331=1072.659,11.503,436.718,173.053,23.460,154.195
C03332=1072.666,11.754,436.704,173.055,23.463,154.196
C03333=1072.672,12.003,436.689,173.057,23.465,154.196
C03334=1072.678,12.252,436.675,173.058,23.468,154.196
C03335=1072.684,12.502,436.660,173.059,23.470,154.196
C03336=1072.690,12.752,436.646,173.061,23.473,154.197
C03337=1072.696,13.001,436.631,173.062,23.475,154.197
C03338=1072.702,13.250,436.616,173.063,23.477,154.197
C03339=1072.708,13.500,436.601,173.064,23.480,154.198
C03340=1072.714,13.749,436.587,173.066,23.483,154.198
C03341=1072.720,13.999,436.572,173.067,23.485,154.198
C03342=1072.726,14.280,436.555,173.069,23.488,154.198
C03343=1072.734,14.560,436.539,173.070,23.491,154.199
C03344=1072.740,14.840,436.522,173.073,23.494,154.199
C03345=1072.747,15.121,436.506,173.074,23.497,154.199
C03346=1072.752,15.371,436.490,173.075,23.499,154.200
C03347=1072.758,15.620,436.476,173.076,23.501,154.200
C03348=1072.765,15.870,436.461,173.078,23.504,154.200
C03349=1072.770,16.119,436.447,173.079,23.507,154.201
C03350=1072.776,16.369,436.431,173.081,23.510,154.201
C03351=1072.782,16.618,436.417,173.082,23.512,154.201
C03352=1072.788,16.868,436.402,173.084,23.514,154.202
C03353=1072.794,17.117,436.387,173.085,23.517,154.202
C03354=1072.799,17.367,436.372,173.086,23.519,154.202
C03355=1072.806,17.616,436.357,173.087,23.522,154.203
C03356=1072.811,17.865,436.342,173.089,23.525,154.203
C03357=1072.818,18.115,436.327,173.090,23.527,154.203
C03358=1072.823,18.364,436.312,173.091,23.529,154.203
C03359=1072.829,18.614,436.297,173.093,23.532,154.204
C03360=1072.836,18.863,436.282,173.095,23.535,154.204
C03361=1072.841,19.113,436.267,173.096,23.538,154.204
C03362=1072.847,19.362,436.252,173.097,23.540,154.205
C03363=1072.853,19.611,436.237,173.099,23.542,154.205
C03364=1072.859,19.861,436.223,173.100,23.545,154.205
C03365=1072.865,20.111,436.207,173.101,23.547,154.205
C03366=1072.871,20.360,436.192,173.102,23.550,154.206
C03367=1072.877,20.610,436.177,173.104,23.553,154.206
C03368=1072.882,20.859,436.162,173.106,23.555,154.206
C03369=1072.889,21.108,436.147,173.107,23.558,154.207
C03370=1072.894,21.358,436.132,173.108,23.560,154.207
C03371=1072.900,21.607,436.117,173.110,23.563,154.207
C03372=1072.906,21.857,436.102,173.111,23.566,154.208
C03373=1072.912,22.107,436.087,173.112,23.568,154.208
C03374=1072.918,22.356,436.072,173.113,23.570,154.208
C03375=1072.923,22.606,436.057,173.115,23.573,154.209
C03376=1072.929,22.855,436.042,173.117,23.576,154.209
C03377=1072.935,23.105,436.026,173.118,23.578,154.209
C03378=1072.941,23.355,436.012,173.119,23.581,154.209
C03379=1072.947,23.604,435.997,173.121,23.583,154.210
C03380=1072.953,23.853,435.981,173.122,23.586,154.210
C03381=1072.959,24.103,435.966,173.123,23.589,154.210
C03382=1072.964,24.352,435.951,173.125,23.591,154.211
C03383=1072.971,24.601,435.936,173.126,23.593,154.211
C03384=1072.977,24.851,435.921,173.128,23.597,154.211
C03385=1072.982,25.100,435.906,173.129,23.599,154.212
C03386=1072.989,25.350,435.891,173.131,23.602,154.212
C03387=1072.995,25.599,435.874,173.132,23.604,154.212
C03388=1073.000,25.848,435.860,173.133,23.606,154.212
C03389=1073.006,26.098,435.844,173.134,23.609,154.213
C03390=1073.012,26.348,435.829,173.136,23.612,154.213
C03391=1073.018,26.598,435.814,173.137,23.614,154.213
C03392=1073.024,26.846,435.798,173.139,23.617,154.214
C03393=1073.030,27.096,435.783,173.140,23.619,154.214
C03394=1073.036,27.346,435.768,173.142,23.622,154.214
C03395=1073.041,27.595,435.753,173.143,23.625,154.215
C03396=1073.048,27.844,435.737,173.144,23.627,154.215
C03397=1073.053,28.094,435.722,173.146,23.629,154.215
C03398=1073.060,28.344,435.707,173.147,23.632,154.216
C03399=1073.065,28.593,435.691,173.148,23.635,154.216
C03400=1073.072,28.842,435.676,173.150,23.638,154.216
C03401=1073.077,29.092,435.660,173.152,23.640,154.216
C03402=1073.083,29.341,435.646,173.153,23.643,154.217
C03403=1073.089,29.590,435.629,173.154,23.645,154.217
C03404=1073.095,29.840,435.614,173.155,23.648,154.217
C03405=1073.101,30.090,435.599,173.157,23.650,154.218
C03406=1073.107,30.372,435.581,173.159,23.653,154.218
C03407=1073.114,30.654,435.564,173.160,23.656,154.219
C03408=1073.120,30.936,435.546,173.161,23.659,154.219
C03409=1073.128,31.217,435.529,173.163,23.662,154.219
C03410=1073.133,31.467,435.514,173.164,23.665,154.220
C03411=1073.139,31.716,435.497,173.166,23.668,154.220
C03412=1073.145,31.966,435.482,173.167,23.670,154.220
C03413=1073.151,32.216,435.467,173.168,23.672,154.220
C03414=1073.156,32.464,435.451,173.170,23.675,154.221
C03415=1073.162,32.714,435.436,173.172,23.678,154.221
C03416=1073.168,32.963,435.420,173.173,23.680,154.221
C03417=1073.174,33.213,435.404,173.174,23.683,154.222
C03418=1073.180,33.462,435.390,173.176,23.686,154.222
C03419=1073.186,33.711,435.373,173.177,23.688,154.222
C03420=1073.191,33.961,435.358,173.178,23.691,154.223
C03421=1073.198,34.210,435.342,173.179,23.694,154.223
C03422=1073.204,34.460,435.327,173.181,23.696,154.223
C03423=1073.209,34.709,435.311,173.183,23.699,154.224
C03424=1073.215,34.959,435.295,173.184,23.701,154.224
C03425=1073.221,35.208,435.280,173.185,23.704,154.224
C03426=1073.227,35.458,435.264,173.187,23.706,154.225
C03427=1073.233,35.707,435.248,173.188,23.709,154.225
C03428=1073.239,35.956,435.233,173.189,23.711,154.225
C03429=1073.245,36.206,435.217,173.190,23.714,154.226
C03430=1073.250,36.456,435.201,173.193,23.717,154.226
C03431=1073.257,36.705,435.186,173.194,23.719,154.226
C03432=1073.263,36.955,435.170,173.195,23.722,154.226
C03433=1073.269,37.204,435.154,173.196,23.725,154.227
C03434=1073.274,37.453,435.139,173.198,23.727,154.227
C03435=1073.280,37.702,435.123,173.199,23.729,154.227
C03436=1073.286,37.952,435.108,173.200,23.732,154.228
C03437=1073.292,38.202,435.091,173.202,23.735,154.228
C03438=1073.298,38.451,435.075,173.204,23.738,154.228
C03439=1073.303,38.701,435.059,173.205,23.740,154.229
C03440=1073.309,38.950,435.044,173.206,23.743,154.229
C03441=1073.315,39.199,435.029,173.208,23.745,154.229
C03442=1073.321,39.449,435.012,173.209,23.748,154.230
C03443=1073.327,39.698,434.996,173.210,23.751,154.230
C03444=1073.333,39.948,434.981,173.211,23.753,154.230
C03445=1073.339,40.197,434.964,173.214,23.756,154.230
C03446=1073.344,40.447,434.949,173.215,23.759,154.231
C03447=1073.350,40.696,434.933,173.216,23.761,154.231
C03448=1073.356,40.945,434.917,173.217,23.764,154.231
C03449=1073.361,41.195,434.901,173.219,23.766,154.232
C03450=1073.367,41.445,434.885,173.220,23.769,154.232
C03451=1073.374,41.694,434.869,173.221,23.771,154.232
C03452=1073.380,41.943,434.853,173.224,23.774,154.233
C03453=1073.385,42.192,434.838,173.225,23.777,154.233
C03454=1073.391,42.442,434.821,173.226,23.779,154.233
C03455=1073.397,42.691,434.805,173.227,23.782,154.234
C03456=1073.402,42.941,434.790,173.229,23.785,154.234
C03457=1073.408,43.190,434.773,173.230,23.787,154.234
C03458=1073.414,43.440,434.757,173.231,23.789,154.235
C03459=1073.420,43.689,434.741,173.233,23.792,154.235
C03460=1073.426,43.939,434.725,173.235,23.795,154.235
C03461=1073.432,44.188,434.709,173.236,23.798,154.236
C03462=1073.437,44.437,434.693,173.237,23.800,154.236
C03463=1073.443,44.686,434.677,173.238,23.803,154.236
C03464=1073.449,44.936,434.661,173.240,23.805,154.237
C03465=1073.455,45.186,434.645,173.241,23.808,154.237
C03466=1073.460,45.435,434.628,173.243,23.811,154.237
C03467=1073.466,45.685,434.612,173.244,23.814,154.238
C03468=1073.472,45.934,434.596,173.246,23.816,154.238
C03469=1073.478,46.183,434.580,173.247,23.819,154.238
C03470=1073.484,46.465,434.562,173.249,23.822,154.239
C03471=1073.491,46.747,434.544,173.250,23.825,154.239
C03472=1073.497,47.029,434.526,173.251,23.828,154.239
C03473=1073.504,47.311,434.507,173.253,23.831,154.240
C03474=1073.510,47.561,434.491,173.255,23.834,154.240
C03475=1073.514,47.810,434.474,173.256,23.836,154.240
C03476=1073.520,48.059,434.458,173.257,23.839,154.241
C03477=1073.526,48.308,434.442,173.259,23.841,154.241
C03478=1073.532,48.558,434.426,173.261,23.845,154.241
C03479=1073.538,48.807,434.409,173.262,23.847,154.242
C03480=1073.544,49.056,434.393,173.263,23.849,154.242
C03481=1073.549,49.306,434.376,173.264,23.852,154.242
C03482=1073.555,49.555,434.360,173.266,23.855,154.243
C03483=1073.561,49.805,434.344,173.267,23.857,154.243
C03484=1073.567,50.055,434.328,173.268,23.860,154.243
C03485=1073.573,50.304,434.312,173.271,23.863,154.244
C03486=1073.579,50.553,434.296,173.272,23.865,154.244
C03487=1073.584,50.803,434.279,173.273,23.868,154.244
C03488=1073.590,51.052,434.263,173.274,23.870,154.245
C03489=1073.596,51.302,434.246,173.276,23.873,154.245
C03490=1073.602,51.551,434.230,173.277,23.876,154.245
C03491=1073.608,51.800,434.214,173.279,23.879,154.246
C03492=1073.613,52.050,434.197,173.280,23.881,154.246
C03493=1073.619,52.299,434.181,173.282,23.884,154.246
C03494=1073.625,52.549,434.164,173.283,23.886,154.247
C03495=1073.631,52.797,434.147,173.284,23.889,154.247
C03496=1073.637,53.047,434.131,173.285,23.892,154.247
C03497=1073.642,53.296,434.114,173.288,23.894,154.248
C03498=1073.648,53.546,434.098,173.289,23.897,154.248
C03499=1073.654,53.795,434.082,173.290,23.900,154.248
C03500=1073.660,54.045,434.066,173.292,23.902,154.249
C03501=1073.666,54.294,434.049,173.293,23.904,154.249
C03502=1073.671,54.544,434.033,173.294,23.907,154.249
C03503=1073.677,54.793,434.016,173.296,23.910,154.249
C03504=1073.683,55.042,434.000,173.298,23.912,154.250
C03505=1073.689,55.292,433.984,173.299,23.915,154.250
C03506=1073.695,55.541,433.966,173.300,23.918,154.250
C03507=1073.701,55.790,433.950,173.301,23.920,154.251
C03508=1073.707,56.039,433.934,173.303,23.923,154.251
C03509=1073.713,56.289,433.917,173.305,23.926,154.251
C03510=1073.718,56.538,433.901,173.306,23.928,154.252
C03511=1073.724,56.788,433.884,173.308,23.931,154.252
C03512=1073.730,57.038,433.868,173.309,23.934,154.252
C03513=1073.737,57.286,433.851,173.310,23.936,154.253
C03514=1073.742,57.536,433.834,173.311,23.938,154.253
C03515=1073.748,57.785,433.818,173.314,23.941,154.253
C03516=1073.754,58.035,433.801,173.315,23.944,154.254
C03517=1073.760,58.284,433.784,173.316,23.946,154.254
C03518=1073.765,58.533,433.768,173.318,23.949,154.254
C03519=1073.771,58.783,433.751,173.319,23.951,154.254
C03520=1073.778,59.033,433.735,173.320,23.954,154.255
C03521=1073.783,59.282,433.718,173.322,23.957,154.255
C03522=1073.789,59.531,433.701,173.324,23.959,154.255
C03523=1073.795,59.780,433.685,173.325,23.962,154.256
C03524=1073.801,60.030,433.668,173.326,23.964,154.256
C03525=1073.807,60.279,433.651,173.328,23.967,154.256
C03526=1073.813,60.528,433.634,173.329,23.969,154.257
C03527=1073.819,60.778,433.618,173.331,23.973,154.257
C03528=1073.824,61.028,433.601,173.332,23.975,154.257
C03529=1073.831,61.277,433.584,173.334,23.977,154.258
C03530=1073.837,61.526,433.568,173.335,23.980,154.258
C03531=1073.842,61.776,433.551,173.336,23.982,154.258
C03532=1073.848,62.024,433.534,173.338,23.985,154.259
C03533=1073.855,62.274,433.517,173.340,23.988,154.259
C03534=1073.861,62.556,433.499,173.341,23.991,154.259
C03535=1073.868,62.838,433.479,173.343,23.993,154.260
C03536=1073.874,63.119,433.460,173.344,23.996,154.260
C03537=1073.882,63.401,433.441,173.346,24.000,154.260
C03538=1073.888,63.650,433.425,173.348,24.002,154.261
C03539=1073.893,63.900,433.408,173.349,24.004,154.261
C03540=1073.899,64.149,433.391,173.350,24.007,154.261
C03541=1073.905,64.398,433.375,173.352,24.009,154.261
C03542=1073.911,64.648,433.357,173.353,24.012,154.262
C03543=1073.916,64.897,433.340,173.355,24.015,154.262
C03544=1073.923,65.146,433.323,173.357,24.017,154.262
C03545=1073.928,65.396,433.306,173.358,24.020,154.263
C03546=1073.934,65.644,433.289,173.359,24.022,154.263
C03547=1073.940,65.895,433.272,173.360,24.025,154.263
C03548=1073.946,66.144,433.256,173.363,24.028,154.264
C03549=1073.951,66.393,433.238,173.364,24.031,154.264
C03550=1073.957,66.643,433.222,173.365,24.033,154.264
C03551=1073.963,66.892,433.204,173.367,24.035,154.265
C03552=1073.969,67.142,433.188,173.368,24.038,154.265
C03553=1073.975,67.391,433.170,173.370,24.041,154.265
C03554=1073.980,67.640,433.153,173.371,24.043,154.266
C03555=1073.986,67.889,433.136,173.373,24.046,154.266
C03556=1073.992,68.138,433.119,173.374,24.049,154.266
C03557=1073.998,68.388,433.102,173.375,24.051,154.267
C03558=1074.004,68.637,433.085,173.377,24.054,154.267
C03559=1074.010,68.887,433.068,173.379,24.057,154.267
C03560=1074.015,69.136,433.051,173.380,24.059,154.268
C03561=1074.021,69.386,433.034,173.381,24.061,154.268
C03562=1074.028,69.635,433.017,173.383,24.064,154.268
C03563=1074.033,69.884,432.999,173.384,24.067,154.268
C03564=1074.038,70.133,432.982,173.386,24.069,154.269
C03565=1074.045,70.382,432.965,173.387,24.072,154.269
C03566=1074.050,70.632,432.948,173.389,24.075,154.269
C03567=1074.056,70.881,432.930,173.390,24.077,154.270
C03568=1074.062,71.130,432.913,173.391,24.080,154.270
C03569=1074.067,71.380,432.897,173.393,24.083,154.270
C03570=1074.073,71.630,432.879,173.395,24.085,154.271
C03571=1074.079,71.879,432.861,173.396,24.088,154.271
C03572=1074.085,72.128,432.845,173.397,24.090,154.271
C03573=1074.090,72.377,432.827,173.399,24.093,154.272
C03574=1074.097,72.627,432.809,173.401,24.096,154.272
C03575=1074.103,72.876,432.793,173.402,24.098,154.272
C03576=1074.108,73.125,432.775,173.404,24.101,154.273
C03577=1074.114,73.375,432.758,173.405,24.103,154.273
C03578=1074.120,73.624,432.740,173.406,24.106,154.273
C03579=1074.125,73.874,432.723,173.408,24.109,154.274
C03580=1074.131,74.122,432.706,173.410,24.111,154.274
C03581=1074.137,74.372,432.688,173.411,24.114,154.274
C03582=1074.143,74.621,432.671,173.412,24.116,154.275
C03583=1074.148,74.871,432.654,173.414,24.119,154.275
C03584=1074.155,75.120,432.636,173.416,24.122,154.275
C03585=1074.160,75.369,432.619,173.417,24.124,154.276
C03586=1074.166,75.618,432.601,173.418,24.127,154.276
C03587=1074.172,75.868,432.583,173.420,24.129,154.276
C03588=1074.177,76.118,432.567,173.422,24.133,154.276
C03589=1074.183,76.366,432.550,173.423,24.135,154.277
C03590=1074.190,76.616,432.532,173.425,24.137,154.277
C03591=1074.195,76.865,432.514,173.426,24.140,154.277
C03592=1074.201,77.114,432.496,173.427,24.143,154.278
C03593=1074.208,77.364,432.479,173.429,24.145,154.278
C03594=1074.213,77.613,432.462,173.431,24.148,154.278
C03595=1074.218,77.862,432.445,173.432,24.150,154.279
C03596=1074.224,78.112,432.427,173.433,24.153,154.279
C03597=1074.230,78.361,432.409,173.436,24.156,154.279
C03598=1074.236,78.643,432.390,173.437,24.159,154.280
C03599=1074.243,78.924,432.370,173.439,24.161,154.280
C03600=1074.249,79.206,432.349,173.440,24.164,154.280
C03601=1074.255,79.487,432.330,173.442,24.167,154.281
C03602=1074.261,79.737,432.312,173.444,24.170,154.281
C03603=1074.267,79.986,432.294,173.445,24.173,154.281
C03604=1074.273,80.235,432.277,173.446,24.175,154.282
C03605=1074.279,80.485,432.259,173.448,24.177,154.282
C03606=1074.284,80.734,432.241,173.450,24.181,154.282
C03607=1074.290,80.983,432.224,173.451,24.183,154.283
C03608=1074.296,81.233,432.206,173.452,24.185,154.283
C03609=1074.301,81.482,432.188,173.454,24.188,154.283
C03610=1074.307,81.732,432.170,173.456,24.191,154.284
C03611=1074.313,81.981,432.153,173.457,24.193,154.284
C03612=1074.318,82.230,432.135,173.458,24.196,154.284
C03613=1074.325,82.479,432.117,173.460,24.199,154.285
C03614=1074.330,82.728,432.100,173.461,24.201,154.285
C03615=1074.336,82.977,432.082,173.463,24.204,154.285
C03616=1074.342,83.227,432.064,173.465,24.207,154.286
C03617=1074.347,83.476,432.047,173.466,24.209,154.286
C03618=1074.353,83.726,432.029,173.467,24.211,154.286
C03619=1074.359,83.975,432.011,173.469,24.215,154.286
C03620=1074.364,84.224,431.993,173.471,24.217,154.287
C03621=1074.371,84.474,431.976,173.472,24.219,154.287
C03622=1074.376,84.723,431.958,173.473,24.222,154.287
C03623=1074.382,84.973,431.940,173.476,24.225,154.288
C03624=1074.388,85.221,431.922,173.477,24.227,154.288
C03625=1074.394,85.471,431.904,173.478,24.230,154.288
C03626=1074.400,85.720,431.886,173.480,24.232,154.289
C03627=1074.406,85.970,431.868,173.482,24.235,154.289
C03628=1074.411,86.219,431.851,173.483,24.238,154.289
C03629=1074.416,86.468,431.833,173.484,24.240,154.290
C03630=1074.422,86.718,431.815,173.486,24.243,154.290
C03631=1074.428,86.966,431.796,173.487,24.245,154.290
C03632=1074.434,87.216,431.778,173.489,24.248,154.290
C03633=1074.440,87.465,431.761,173.491,24.251,154.291
C03634=1074.446,87.715,431.743,173.492,24.253,154.291
C03635=1074.451,87.964,431.725,173.493,24.256,154.291
C03636=1074.458,88.213,431.707,173.496,24.259,154.292
C03637=1074.463,88.462,431.689,173.497,24.261,154.292
C03638=1074.469,88.712,431.671,173.498,24.263,154.292
C03639=1074.475,88.961,431.654,173.500,24.266,154.293
